KUKA KRL program: MyProgram_043().src

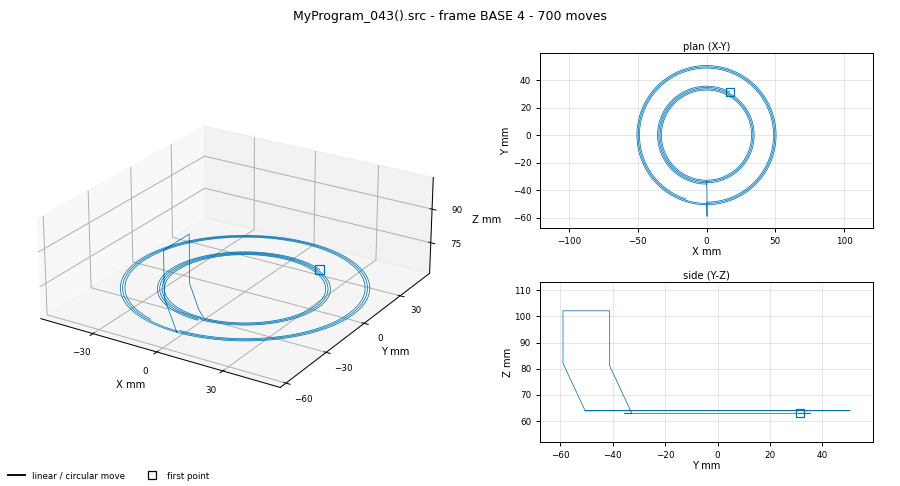
[picture p0: tool path of MyProgram_043().src in frame BASE 4, 700 of 700 moves have a stored position in this frame; points joined in program order, loops and branches not executed]
&ACCESS RVP
&REL 1
&PARAM TEMPLATE = C:\KRC\Roboter\Template\vorgabe
&PARAM EDITMASK = *
DEF MyProgram_043()
; ---- Setting reference (Base) ----
$BASE = BASE_DATA[4]

; --------------------------
; ---- Setting tool (TCP) ----
$TOOL = TOOL_DATA[3]
; --------------------------

$VEL.CP = VEL_APROX_PRINT
Startdeposition()
$VEL.CP = VEL_PRINT
LIN {X 16.8106,Y 31.3623,Z 63,A 55.0219,B 24.8198,C -3.0966,E1 25.0743,E2 -332.082} C_DIS
LIN {X 15.1626,Y 32.1914,Z 63,A 58.444,B 24.8186,C -3.1061,E1 25.0657,E2 -335.5177} C_DIS
LIN {X 13.6863,Y 32.8466,Z 63,A 60.9458,B 24.8184,C -3.1075,E1 25.0593,E2 -338.0168} C_DIS
LIN {X 11.5604,Y 33.654,Z 63,A 64.6472,B 24.818,C -3.1112,E1 25.0495,E2 -341.7194} C_DIS
LIN {X 8.9536,Y 34.4389,Z 63,A 68.8262,B 24.818,C -3.1115,E1 25.0383,E2 -345.8923} C_DIS
LIN {X 7.0657,Y 34.8749,Z 63,A 72.0407,B 24.8177,C -3.1142,E1 25.0295,E2 -349.1089} C_DIS
LIN {X 4.955,Y 35.237,Z 63,A 75.0597,B 24.8182,C -3.1099,E1 25.0213,E2 -352.1148} C_DIS
LIN {X 3.7288,Y 35.3877,Z 63,A 77.2434,B 24.8178,C -3.1126,E1 25.0152,E2 -354.3034} C_DIS
LIN {X 2.076,Y 35.5232,Z 63,A 79.8681,B 24.8179,C -3.1121,E1 25.0079,E2 -356.9257} C_DIS
LIN {X 0.3777,Y 35.582,Z 63,A 82.8072,B 24.8177,C -3.1142,E1 24.9997,E2 -359.8692} C_DIS
LIN {X -1.1222,Y 35.5659,Z 63,A 85.2424,B 24.8177,C -3.1138,E1 24.9929,E2 -362.3038} C_DIS
LIN {X -2.9049,Y 35.4649,Z 63,A 88.7717,B 24.817,C -3.1201,E1 24.983,E2 -365.8497} C_DIS
LIN {X -6.81,Y 34.926,Z 63,A 94.1207,B 24.8188,C -3.1045,E1 24.9683,E2 -371.1662} C_DIS
LIN {X -9.2966,Y 34.3477,Z 63,A 99.2069,B 24.818,C -3.1114,E1 24.9545,E2 -376.276} C_DIS
LIN {X -11.642,Y 33.6256,Z 63,A 102.3463,B 24.8196,C -3.098,E1 24.9462,E2 -379.3892} C_DIS
LIN {X -13.5299,Y 32.9112,Z 63,A 106.2069,B 24.8193,C -3.1002,E1 24.9362,E2 -383.2634} C_DIS
LIN {X -15.9173,Y 31.8253,Z 63,A 110.4655,B 24.82,C -3.0941,E1 24.9255,E2 -387.5184} C_DIS
LIN {X -18.0289,Y 30.6783,Z 63,A 114.2931,B 24.8208,C -3.087,E1 24.9162,E2 -391.3404} C_DIS
LIN {X -20.7669,Y 28.8954,Z 63,A 118.9134,B 24.8228,C -3.0705,E1 24.9056,E2 -395.9367} C_DIS
LIN {X -22.22,Y 27.7939,Z 63,A 122.3158,B 24.8229,C -3.069,E1 24.898,E2 -399.348} C_DIS
LIN {X -24.1802,Y 26.1054,Z 63,A 126.2379,B 24.8243,C -3.0574,E1 24.8899,E2 -403.2579} C_DIS
LIN {X -25.3409,Y 24.9807,Z 63,A 128.7227,B 24.8251,C -3.0502,E1 24.885,E2 -405.7359} C_DIS
LIN {X -26.8356,Y 23.3676,Z 63,A 133.3079,B 24.825,C -3.0515,E1 24.8764,E2 -410.3446} C_DIS
LIN {X -28.8287,Y 20.86,Z 63,A 137.8819,B 24.8271,C -3.0325,E1 24.8687,E2 -414.895} C_DIS
LIN {X -30.1785,Y 18.8534,Z 63,A 141.3427,B 24.8288,C -3.0179,E1 24.8635,E2 -418.3383} C_DIS
LIN {X -31.0448,Y 17.3901,Z 63,A 144.4056,B 24.8293,C -3.0132,E1 24.8592,E2 -421.4059} C_DIS
LIN {X -31.9505,Y 15.6632,Z 63,A 147.8398,B 24.8301,C -3.0068,E1 24.8549,E2 -424.8432} C_DIS
LIN {X -33.01,Y 13.2873,Z 63,A 152.0346,B 24.8315,C -2.9945,E1 24.8503,E2 -429.0318} C_DIS
LIN {X -33.7447,Y 11.2915,Z 63,A 155.0687,B 24.833,C -2.9806,E1 24.8475,E2 -432.0499} C_DIS
LIN {X -34.2032,Y 9.8157,Z 63,A 157.7943,B 24.8336,C -2.9752,E1 24.8454,E2 -434.7782} C_DIS
LIN {X -34.7895,Y 7.4763,Z 63,A 161.2013,B 24.8355,C -2.959,E1 24.8432,E2 -438.1663} C_DIS
LIN {X -35.0815,Y 5.9572,Z 63,A 164.5571,B 24.8355,C -2.9589,E1 24.8415,E2 -441.5418} C_DIS
LIN {X -35.4137,Y 3.4768,Z 63,A 168.3045,B 24.8372,C -2.9437,E1 24.8403,E2 -445.2754} C_DIS
LIN {X -35.5404,Y 1.7652,Z 63,A 171.2528,B 24.8379,C -2.9367,E1 24.8399,E2 -448.2247} C_DIS
LIN {X -35.5745,Y -0.8093,Z 63,A 174.7396,B 24.84,C -2.9179,E1 24.8399,E2 -451.6875} C_DIS
LIN {X -35.5121,Y -2.2598,Z 63,A 177.4397,B 24.8405,C -2.9139,E1 24.8402,E2 -454.3941} C_DIS
LIN {X -35.3438,Y -4.1241,Z 63,A -179.4444,B 24.8414,C -2.9055,E1 24.8411,E2 -457.5085} C_DIS
LIN {X -35.0507,Y -6.1346,Z 63,A -175.5471,B 24.8419,C -2.9011,E1 24.8429,E2 -461.4187} C_DIS
LIN {X -34.3748,Y -9.1965,Z 63,A -171.0715,B 24.8441,C -2.8808,E1 24.8458,E2 -465.8718} C_DIS
LIN {X -33.7609,Y -11.2432,Z 63,A -168.1618,B 24.8457,C -2.866,E1 24.8482,E2 -468.7628} C_DIS
LIN {X -33.2462,Y -12.6842,Z 63,A -165.0655,B 24.8458,C -2.8647,E1 24.8512,E2 -471.8735} C_DIS
LIN {X -32.3646,Y -14.7906,Z 63,A -161.0277,B 24.8466,C -2.8578,E1 24.8558,E2 -475.9171} C_DIS
LIN {X -31.2752,Y -16.9722,Z 63,A -157.1273,B 24.8477,C -2.8471,E1 24.8608,E2 -479.8126} C_DIS
LIN {X -30.1984,Y -18.8215,Z 63,A -153.4943,B 24.8485,C -2.8401,E1 24.8661,E2 -483.4474} C_DIS
LIN {X -28.8099,Y -20.8856,Z 63,A -150.0856,B 24.8501,C -2.8246,E1 24.8715,E2 -486.8358} C_DIS
LIN {X -27.7664,Y -22.253,Z 63,A -147.0838,B 24.8506,C -2.8204,E1 24.8767,E2 -489.8417} C_DIS
LIN {X -26.3842,Y -23.8768,Z 63,A -143.5764,B 24.8513,C -2.8135,E1 24.8832,E2 -493.3486} C_DIS
LIN {X -24.5192,Y -25.787,Z 63,A -139.4733,B 24.8524,C -2.8028,E1 24.8913,E2 -497.4433} C_DIS
LIN {X -23.1525,Y -27.0216,Z 63,A -136.4644,B 24.853,C -2.7976,E1 24.8976,E2 -500.4517} C_DIS
LIN {X -21.8431,Y -28.0903,Z 63,A -133.742,B 24.8535,C -2.7928,E1 24.9036,E2 -503.1727} C_DIS
LIN {X -20.5207,Y -29.0711,Z 63,A -130.4876,B 24.8533,C -2.7948,E1 24.911,E2 -506.4432} C_DIS
LIN {X -18.3593,Y -30.4819,Z 63,A -126.8445,B 24.8545,C -2.7832,E1 24.9196,E2 -510.0701} C_DIS
LIN {X -16.5344,Y -31.5089,Z 63,A -123.3892,B 24.8549,C -2.7797,E1 24.9281,E2 -513.5269} C_DIS
LIN {X -14.4801,Y -32.5045,Z 63,A -119.6559,B 24.8552,C -2.7763,E1 24.9375,E2 -517.2613} C_DIS
LIN {X -12.1069,Y -33.4608,Z 63,A -115.6723,B 24.8558,C -2.771,E1 24.9479,E2 -521.2407} C_DIS
LIN {X -10.7396,Y -33.9249,Z 63,A -113.2876,B 24.8558,C -2.7699,E1 24.9542,E2 -523.6272} C_DIS
LIN {X -8.9212,Y -34.4472,Z 63,A -110.3502,B 24.8562,C -2.7668,E1 24.9621,E2 -526.5618} C_DIS
LIN {X -7.1974,Y -34.8481,Z 63,A -107.4065,B 24.8562,C -2.7666,E1 24.9702,E2 -529.5087} C_DIS
LIN {X -5.1932,Y -35.2031,Z 63,A -104.0844,B 24.8562,C -2.7663,E1 24.9793,E2 -532.833} C_DIS
LIN {X -3.2172,Y -35.4379,Z 63,A -100.9818,B 24.8564,C -2.7647,E1 24.988,E2 -535.9337} C_DIS
LIN {X -1.3671,Y -35.5576,Z 63,A -98.1082,B 24.8565,C -2.7636,E1 24.996,E2 -538.8052} C_DIS
LIN {X 0.1757,Y -35.5825,Z 63,A -95.5141,B 24.8564,C -2.7655,E1 25.0032,E2 -541.4039} C_DIS
Enddeposition()
LIN {X 0.1757,Y -35.5825,Z 63,A -95.5141,B 24.8564,C -2.7655,E1 25.0032,E2 -541.4039} C_DIS
Startdeposition()
$VEL.CP = VEL_PRINT
LIN {X -0.0635,Y -34.634,Z 63,A -97.3781,B 24.8565,C -2.764,E1 24.998,E2 -539.5365} C_DIS
LIN {X -1.8941,Y -34.5819,Z 63,A -100.1272,B 24.8562,C -2.767,E1 24.9904,E2 -536.7939} C_DIS
LIN {X -3.4007,Y -34.467,Z 63,A -102.9968,B 24.8566,C -2.7628,E1 24.9823,E2 -533.9131} C_DIS
LIN {X -5.0318,Y -34.2667,Z 63,A -105.5259,B 24.8563,C -2.7655,E1 24.9754,E2 -531.3884} C_DIS
LIN {X -6.3765,Y -34.0415,Z 63,A -107.7692,B 24.8563,C -2.7664,E1 24.9692,E2 -529.1449} C_DIS
LIN {X -7.847,Y -33.7331,Z 63,A -110.4703,B 24.8563,C -2.7651,E1 24.9618,E2 -526.4375} C_DIS
LIN {X -10.2211,Y -33.0912,Z 63,A -113.9954,B 24.8555,C -2.7736,E1 24.9524,E2 -522.927} C_DIS
LIN {X -12.797,Y -32.1832,Z 63,A -119.1428,B 24.8558,C -2.7708,E1 24.9388,E2 -517.7624} C_DIS
LIN {X -14.7742,Y -31.325,Z 63,A -122.8072,B 24.8555,C -2.7736,E1 24.9295,E2 -514.0959} C_DIS
LIN {X -16.8249,Y -30.2725,Z 63,A -126.1313,B 24.8545,C -2.7834,E1 24.9213,E2 -510.7859} C_DIS
LIN {X -18.706,Y -29.1476,Z 63,A -130.3212,B 24.8545,C -2.783,E1 24.9113,E2 -506.5821} C_DIS
LIN {X -20.4124,Y -27.9792,Z 63,A -133.6933,B 24.8539,C -2.7891,E1 24.9037,E2 -503.2128} C_DIS
LIN {X -22.2197,Y -26.5668,Z 63,A -137.5576,B 24.8532,C -2.7952,E1 24.8953,E2 -499.3487} C_DIS
LIN {X -23.9602,Y -25.0084,Z 63,A -141.3526,B 24.8524,C -2.8035,E1 24.8875,E2 -495.5579} C_DIS
LIN {X -25.5766,Y -23.3526,Z 63,A -145.1707,B 24.8515,C -2.8117,E1 24.8802,E2 -491.7428} C_DIS
LIN {X -27.0497,Y -21.6299,Z 63,A -148.7189,B 24.8504,C -2.822,E1 24.8739,E2 -488.2029} C_DIS
LIN {X -28.2319,Y -20.0614,Z 63,A -152.2011,B 24.8498,C -2.8277,E1 24.8681,E2 -484.7175} C_DIS
LIN {X -29.5519,Y -18.0607,Z 63,A -155.8174,B 24.8484,C -2.8408,E1 24.8627,E2 -481.1142} C_DIS
LIN {X -30.3461,Y -16.6929,Z 63,A -159.348,B 24.8485,C -2.8396,E1 24.8578,E2 -477.5623} C_DIS
LIN {X -31.6295,Y -14.1099,Z 63,A -163.645,B 24.8467,C -2.8568,E1 24.8527,E2 -473.283} C_DIS
LIN {X -32.4602,Y -12.0779,Z 63,A -167.3733,B 24.8456,C -2.8662,E1 24.849,E2 -469.5563} C_DIS
LIN {X -33.016,Y -10.4631,Z 63,A -169.9052,B 24.8445,C -2.8769,E1 24.8468,E2 -467.0355} C_DIS
LIN {X -33.6352,Y -8.2566,Z 63,A -173.5321,B 24.8431,C -2.8896,E1 24.8441,E2 -463.4178} C_DIS
LIN {X -34.0004,Y -6.5934,Z 63,A -176.7425,B 24.8425,C -2.8948,E1 24.8423,E2 -460.201} C_DIS
LIN {X -34.2819,Y -4.9246,Z 63,A -179.5712,B 24.8416,C -2.9031,E1 24.8411,E2 -457.3753} C_DIS
LIN {X -34.5211,Y -2.7908,Z 63,A 176.9771,B 24.8403,C -2.9149,E1 24.8402,E2 -453.9312} C_DIS
LIN {X -34.6169,Y -1.0818,Z 63,A 174.3178,B 24.8392,C -2.9251,E1 24.8398,E2 -451.2804} C_DIS
LIN {X -34.6257,Y 0.7559,Z 63,A 170.7594,B 24.8386,C -2.9304,E1 24.8399,E2 -447.7131} C_DIS
LIN {X -34.5394,Y 2.5589,Z 63,A 168.2461,B 24.8372,C -2.9436,E1 24.8403,E2 -445.2163} C_DIS
LIN {X -34.342,Y 4.4866,Z 63,A 164.6999,B 24.8364,C -2.9508,E1 24.8415,E2 -441.6662} C_DIS
LIN {X -33.9758,Y 6.7211,Z 63,A 160.8095,B 24.8352,C -2.9613,E1 24.8434,E2 -437.7778} C_DIS
LIN {X -33.5133,Y 8.7391,Z 63,A 157.8409,B 24.8336,C -2.9756,E1 24.8453,E2 -434.8262} C_DIS
LIN {X -33.034,Y 10.4054,Z 63,A 154.5657,B 24.833,C -2.981,E1 24.848,E2 -431.5449} C_DIS
LIN {X -32.5136,Y 11.9319,Z 63,A 151.8111,B 24.8322,C -2.9883,E1 24.8505,E2 -428.7923} C_DIS
LIN {X -31.6838,Y 13.9879,Z 63,A 148.0384,B 24.831,C -2.9983,E1 24.8547,E2 -425.0225} C_DIS
LIN {X -30.8835,Y 15.6751,Z 63,A 144.9909,B 24.83,C -3.0075,E1 24.8584,E2 -421.9808} C_DIS
LIN {X -29.5734,Y 18.0254,Z 63,A 140.5667,B 24.8285,C -3.0203,E1 24.8646,E2 -417.564} C_DIS
LIN {X -28.3146,Y 19.9454,Z 63,A 136.653,B 24.8275,C -3.0295,E1 24.8707,E2 -413.653} C_DIS
LIN {X -26.9355,Y 21.771,Z 63,A 132.7973,B 24.8264,C -3.0387,E1 24.8774,E2 -409.801} C_DIS
LIN {X -25.4787,Y 23.4593,Z 63,A 129.2123,B 24.8253,C -3.0487,E1 24.884,E2 -406.2238} C_DIS
LIN {X -23.5824,Y 25.3655,Z 63,A 124.6722,B 24.8242,C -3.0581,E1 24.8931,E2 -401.6875} C_DIS
LIN {X -21.8898,Y 26.8393,Z 63,A 121.035,B 24.8232,C -3.0669,E1 24.9008,E2 -398.0572} C_DIS
LIN {X -20.1572,Y 28.1636,Z 63,A 117.5628,B 24.8222,C -3.0754,E1 24.9086,E2 -394.593} C_DIS
LIN {X -18.4097,Y 29.3358,Z 63,A 113.9792,B 24.8215,C -3.0809,E1 24.917,E2 -391.011} C_DIS
LIN {X -16.9995,Y 30.1747,Z 63,A 111.1515,B 24.8211,C -3.0846,E1 24.9238,E2 -388.1835} C_DIS
LIN {X -14.7244,Y 31.3481,Z 63,A 106.2891,B 24.8211,C -3.085,E1 24.9361,E2 -383.3096} C_DIS
LIN {X -11.4307,Y 32.6931,Z 63,A 101.432,B 24.819,C -3.103,E1 24.9486,E2 -378.4851} C_DIS
LIN {X -9.8087,Y 33.2158,Z 63,A 97.9102,B 24.8194,C -3.0989,E1 24.9581,E2 -374.9474} C_DIS
LIN {X -7.2365,Y 33.8696,Z 63,A 94.0249,B 24.8184,C -3.1082,E1 24.9686,E2 -371.0789} C_DIS
LIN {X -5.3631,Y 34.2161,Z 63,A 90.7464,B 24.8183,C -3.1091,E1 24.9776,E2 -367.7995} C_DIS
LIN {X -3.651,Y 34.4408,Z 63,A 87.6697,B 24.8183,C -3.1083,E1 24.9861,E2 -364.7188} C_DIS
LIN {X -2.1391,Y 34.568,Z 63,A 85.0882,B 24.8183,C -3.1085,E1 24.9933,E2 -362.1369} C_DIS
LIN {X 0.4092,Y 34.6319,Z 63,A 81.0243,B 24.818,C -3.1111,E1 25.0047,E2 -358.0793} C_DIS
LIN {X 1.9136,Y 34.5809,Z 63,A 78.6706,B 24.8178,C -3.1128,E1 25.0112,E2 -355.7303} C_DIS
LIN {X 3.832,Y 34.4215,Z 63,A 75.4828,B 24.8178,C -3.1124,E1 25.0201,E2 -352.5435} C_DIS
LIN {X 5.4581,Y 34.2012,Z 63,A 72.8563,B 24.8178,C -3.1127,E1 25.0273,E2 -349.9201} C_DIS
LIN {X 7.3944,Y 33.8352,Z 63,A 69.2492,B 24.8185,C -3.1072,E1 25.0372,E2 -346.3043} C_DIS
LIN {X 10.0204,Y 33.153,Z 63,A 64.8238,B 24.8187,C -3.105,E1 25.0491,E2 -341.8811} C_DIS
LIN {X 12.2173,Y 32.4074,Z 63,A 61.1221,B 24.8189,C -3.1034,E1 25.0588,E2 -338.183} C_DIS
LIN {X 14.2169,Y 31.5813,Z 63,A 57.0676,B 24.8201,C -3.0937,E1 25.0692,E2 -334.1152} C_DIS
LIN {X 16.87,Y 30.2473,Z 63,A 52.6482,B 24.8201,C -3.0936,E1 25.0801,E2 -329.7081} C_DIS
LIN {X 19.2374,Y 28.8,Z 63,A 48.2364,B 24.8206,C -3.089,E1 25.0905,E2 -325.2996} C_DIS
LIN {X 20.4873,Y 27.9243,Z 63,A 45.9769,B 24.8206,C -3.0883,E1 25.0957,E2 -323.0463} C_DIS
LIN {X 21.9684,Y 26.7745,Z 63,A 41.9109,B 24.8228,C -3.07,E1 25.1046,E2 -318.9521} C_DIS
LIN {X 23.9141,Y 25.0527,Z 63,A 37.7836,B 24.8235,C -3.0637,E1 25.113,E2 -314.8268} C_DIS
LIN {X 25.8678,Y 23.0296,Z 63,A 33.4254,B 24.8242,C -3.0577,E1 25.1213,E2 -310.4734} C_DIS
LIN {X 27.3526,Y 21.245,Z 63,A 29.6291,B 24.8252,C -3.0494,E1 25.1279,E2 -306.6751} C_DIS
LIN {X 28.3512,Y 19.893,Z 63,A 26.7406,B 24.8261,C -3.0412,E1 25.1326,E2 -303.7812} C_DIS
LIN {X 29.6598,Y 17.8833,Z 63,A 22.8855,B 24.8271,C -3.0326,E1 25.1383,E2 -299.9253} C_DIS
LIN {X 30.7733,Y 15.891,Z 63,A 19.1935,B 24.8281,C -3.0238,E1 25.1432,E2 -296.2318} C_DIS
LIN {X 31.7469,Y 13.8432,Z 63,A 16.033,B 24.8284,C -3.0219,E1 25.1469,E2 -293.0839} C_DIS
LIN {X 32.5142,Y 11.9303,Z 63,A 12.5189,B 24.8296,C -3.0107,E1 25.1505,E2 -289.5627} C_DIS
LIN {X 33.2079,Y 9.8352,Z 63,A 8.8585,B 24.8309,C -2.9999,E1 25.1536,E2 -285.8975} C_DIS
LIN {X 33.811,Y 7.5051,Z 63,A 4.497,B 24.8328,C -2.9825,E1 25.1565,E2 -281.5201} C_DIS
LIN {X 34.1619,Y 5.6977,Z 63,A 1.4153,B 24.8339,C -2.9727,E1 25.158,E2 -278.4332} C_DIS
LIN {X 34.5054,Y 2.9862,Z 63,A -3.0553,B 24.8354,C -2.9595,E1 25.1594,E2 -273.9578} C_DIS
LIN {X 34.6255,Y 0.7666,Z 63,A -6.5632,B 24.8364,C -2.9505,E1 25.1598,E2 -270.4494} C_DIS
LIN {X 34.5993,Y -1.5455,Z 63,A -10.4486,B 24.8378,C -2.9376,E1 25.1595,E2 -266.5566} C_DIS
LIN {X 34.4732,Y -3.3318,Z 63,A -12.9537,B 24.8381,C -2.935,E1 25.1589,E2 -264.0603} C_DIS
LIN {X 34.2793,Y -4.9431,Z 63,A -16.0017,B 24.8396,C -2.9213,E1 25.1578,E2 -260.9978} C_DIS
LIN {X 33.8998,Y -7.0921,Z 63,A -19.8009,B 24.8412,C -2.9073,E1 25.1558,E2 -257.1876} C_DIS
LIN {X 33.1911,Y -9.892,Z 63,A -24.2794,B 24.8423,C -2.897,E1 25.1525,E2 -252.7104} C_DIS
LIN {X 32.5177,Y -11.9206,Z 63,A -27.8522,B 24.8435,C -2.8857,E1 25.1492,E2 -249.1311} C_DIS
LIN {X 31.6889,Y -13.9762,Z 63,A -32.0187,B 24.8455,C -2.8676,E1 25.1446,E2 -244.9446} C_DIS
LIN {X 30.2023,Y -16.9506,Z 63,A -36.82,B 24.8461,C -2.8619,E1 25.1384,E2 -240.155} C_DIS
LIN {X 29.1784,Y -18.6581,Z 63,A -40.1878,B 24.8472,C -2.8516,E1 25.1335,E2 -236.7801} C_DIS
LIN {X 28.0786,Y -20.2752,Z 63,A -43.5148,B 24.8483,C -2.8416,E1 25.1281,E2 -233.4457} C_DIS
LIN {X 26.632,Y -22.1413,Z 63,A -47.8274,B 24.85,C -2.8259,E1 25.1205,E2 -229.1157} C_DIS
LIN {X 24.3949,Y -24.5844,Z 63,A -52.6985,B 24.8505,C -2.8211,E1 25.1112,E2 -224.2544} C_DIS
LIN {X 23.0523,Y -25.8475,Z 63,A -56.3973,B 24.8522,C -2.8052,E1 25.1035,E2 -220.5329} C_DIS
LIN {X 20.172,Y -28.153,Z 63,A -61.9593,B 24.8527,C -2.7999,E1 25.0912,E2 -214.9785} C_DIS
LIN {X 18.897,Y -29.0233,Z 63,A -64.7157,B 24.8535,C -2.7923,E1 25.0847,E2 -212.2132} C_DIS
LIN {X 16.4975,Y -30.4521,Z 63,A -68.7587,B 24.8535,C -2.7918,E1 25.075,E2 -208.1813} C_DIS
LIN {X 14.7635,Y -31.3299,Z 63,A -72.2932,B 24.8546,C -2.7825,E1 25.0661,E2 -204.6341} C_DIS
LIN {X 12.7079,Y -32.2182,Z 63,A -75.5559,B 24.8546,C -2.783,E1 25.0577,E2 -201.3803} C_DIS
LIN {X 10.6503,Y -32.9556,Z 63,A -79.8648,B 24.8559,C -2.7697,E1 25.0462,E2 -197.0483} C_DIS
LIN {X 8.7345,Y -33.5145,Z 63,A -82.4668,B 24.8553,C -2.7751,E1 25.0393,E2 -194.4632} C_DIS
LIN {X 7.1379,Y -33.8907,Z 63,A -85.5521,B 24.8561,C -2.768,E1 25.0308,E2 -191.3652} C_DIS
LIN {X 5.4364,Y -34.2044,Z 63,A -88.2199,B 24.8561,C -2.7682,E1 25.0235,E2 -188.7007} C_DIS
LIN {X 3.6386,Y -34.4421,Z 63,A -90.8735,B 24.8558,C -2.7706,E1 25.0162,E2 -186.0549} C_DIS
LIN {X 1.5293,Y -34.6,Z 63,A -95.3139,B 24.8571,C -2.7579,E1 25.0037,E2 -181.5861} C_DIS
LIN {X 1.5293,Y -34.6,Z 63,A -95.3139,B 24.8571,C -2.7579,E1 25.0037,E2 -181.5861} C_DIS
Enddeposition()
LIN {X 0.1418,Y -33.6777,Z 63,A -95.815,B 24.8533,C -2.7949,E1 25.0026,E2 -181.1731} C_DIS
Startdeposition()
$VEL.CP = VEL_PRINT
LIN {X 2.8514,Y -33.5634,Z 63,A -91.0405,B 24.8529,C -2.7986,E1 25.0159,E2 -185.9545} C_DIS
LIN {X 4.8668,Y -33.3307,Z 63,A -86.734,B 24.8515,C -2.8113,E1 25.0279,E2 -190.2875} C_DIS
LIN {X 7.9983,Y -32.7205,Z 63,A -81.8757,B 24.8518,C -2.809,E1 25.0411,E2 -195.134} C_DIS
LIN {X 10.4669,Y -32.0159,Z 63,A -77.9995,B 24.8519,C -2.8077,E1 25.0514,E2 -199.0004} C_DIS
LIN {X 11.957,Y -31.4903,Z 63,A -75.0907,B 24.8512,C -2.814,E1 25.0591,E2 -201.918} C_DIS
LIN {X 13.8798,Y -30.6914,Z 63,A -71.4979,B 24.8506,C -2.8198,E1 25.0683,E2 -205.5159} C_DIS
LIN {X 15.8468,Y -29.724,Z 63,A -67.6662,B 24.8498,C -2.8272,E1 25.0778,E2 -209.3547} C_DIS
LIN {X 17.6483,Y -28.6905,Z 63,A -64.1441,B 24.8492,C -2.8334,E1 25.0863,E2 -212.8807} C_DIS
LIN {X 19.2803,Y -27.6203,Z 63,A -60.9493,B 24.8487,C -2.8382,E1 25.0937,E2 -216.076} C_DIS
LIN {X 21.0567,Y -26.2918,Z 63,A -56.8255,B 24.8473,C -2.8509,E1 25.1028,E2 -220.2147} C_DIS
LIN {X 22.9024,Y -24.7006,Z 63,A -53.0751,B 24.8469,C -2.8548,E1 25.1106,E2 -223.9594} C_DIS
LIN {X 24.8683,Y -22.7196,Z 63,A -47.5228,B 24.8444,C -2.8776,E1 25.1213,E2 -229.5416} C_DIS
LIN {X 26.6927,Y -20.5452,Z 63,A -43.482,B 24.8443,C -2.8789,E1 25.1283,E2 -233.5666} C_DIS
LIN {X 28.2034,Y -18.416,Z 63,A -39.1453,B 24.8431,C -2.8895,E1 25.1352,E2 -237.907} C_DIS
LIN {X 29.378,Y -16.4786,Z 63,A -35.0709,B 24.8416,C -2.9035,E1 25.1409,E2 -241.9934} C_DIS
LIN {X 30.309,Y -14.6949,Z 63,A -31.8725,B 24.8409,C -2.9102,E1 25.1449,E2 -245.1907} C_DIS
LIN {X 31.2078,Y -12.6761,Z 63,A -28.104,B 24.8396,C -2.9214,E1 25.1491,E2 -248.9652} C_DIS
LIN {X 31.9406,Y -10.6963,Z 63,A -24.5863,B 24.8385,C -2.9312,E1 25.1523,E2 -252.4863} C_DIS
LIN {X 32.5772,Y -8.5655,Z 63,A -20.7114,B 24.8371,C -2.9442,E1 25.1552,E2 -256.3697} C_DIS
LIN {X 33.1042,Y -6.2243,Z 63,A -17.2808,B 24.8367,C -2.9474,E1 25.1572,E2 -259.7879} C_DIS
LIN {X 33.3154,Y -4.9723,Z 63,A -14.6256,B 24.8352,C -2.9613,E1 25.1584,E2 -262.4605} C_DIS
LIN {X 33.5534,Y -2.9655,Z 63,A -11.342,B 24.8342,C -2.9699,E1 25.1593,E2 -265.7449} C_DIS
LIN {X 33.6455,Y -1.6171,Z 63,A -8.8611,B 24.8331,C -2.9798,E1 25.1597,E2 -268.2345} C_DIS
LIN {X 33.6833,Y 0.1825,Z 63,A -5.9247,B 24.8323,C -2.9875,E1 25.1597,E2 -271.1718} C_DIS
LIN {X 33.6079,Y 2.2618,Z 63,A -2.4105,B 24.8311,C -2.9982,E1 25.1592,E2 -274.6902} C_DIS
LIN {X 33.4146,Y 4.2515,Z 63,A 0.9106,B 24.83,C -3.0075,E1 25.1582,E2 -278.0138} C_DIS
LIN {X 33.1059,Y 6.2155,Z 63,A 4.3752,B 24.8287,C -3.019,E1 25.1566,E2 -281.4854} C_DIS
LIN {X 32.4377,Y 9.0783,Z 63,A 9.8301,B 24.8262,C -3.0405,E1 25.1528,E2 -286.9597} C_DIS
LIN {X 31.5027,Y 11.9242,Z 63,A 14.2081,B 24.8257,C -3.0449,E1 25.1488,E2 -291.3234} C_DIS
LIN {X 30.9466,Y 13.302,Z 63,A 17.0215,B 24.8244,C -3.056,E1 25.1457,E2 -294.1478} C_DIS
LIN {X 30.0175,Y 15.2827,Z 63,A 20.6762,B 24.8234,C -3.0652,E1 25.1412,E2 -297.8046} C_DIS
LIN {X 28.9182,Y 17.2733,Z 63,A 24.9412,B 24.8216,C -3.0808,E1 25.1352,E2 -302.0848} C_DIS
LIN {X 27.6714,Y 19.2068,Z 63,A 28.1622,B 24.8216,C -3.0809,E1 25.1302,E2 -305.29} C_DIS
LIN {X 26.5354,Y 20.7488,Z 63,A 31.6472,B 24.8203,C -3.0917,E1 25.1243,E2 -308.784} C_DIS
LIN {X 25.1034,Y 22.4594,Z 63,A 35.6666,B 24.8189,C -3.1033,E1 25.1169,E2 -312.8127} C_DIS
LIN {X 23.582,Y 24.0522,Z 63,A 39.1309,B 24.8185,C -3.1072,E1 25.1101,E2 -316.2717} C_DIS
LIN {X 21.9707,Y 25.5328,Z 63,A 42.8867,B 24.8176,C -3.1148,E1 25.1023,E2 -320.0305} C_DIS
LIN {X 20.2752,Y 26.8985,Z 63,A 46.865,B 24.8164,C -3.125,E1 25.0935,E2 -324.0183} C_DIS
LIN {X 17.948,Y 28.504,Z 63,A 51.2457,B 24.8162,C -3.1269,E1 25.0833,E2 -328.3891} C_DIS
LIN {X 16.1698,Y 29.5493,Z 63,A 54.8034,B 24.8155,C -3.1323,E1 25.0746,E2 -331.9491} C_DIS
LIN {X 14.4618,Y 30.4217,Z 63,A 57.51,B 24.8159,C -3.1293,E1 25.0679,E2 -334.6412} C_DIS
LIN {X 13.009,Y 31.0705,Z 63,A 60.7616,B 24.8147,C -3.139,E1 25.0595,E2 -337.9079} C_DIS
LIN {X 10.9037,Y 31.8707,Z 63,A 64.6332,B 24.8143,C -3.1428,E1 25.0494,E2 -341.7807} C_DIS
LIN {X 8.7457,Y 32.5288,Z 63,A 68.6978,B 24.8136,C -3.1481,E1 25.0384,E2 -345.8512} C_DIS
LIN {X 6.1905,Y 33.1107,Z 63,A 72.9035,B 24.8138,C -3.1471,E1 25.027,E2 -350.0492} C_DIS
LIN {X 3.9481,Y 33.4518,Z 63,A 76.7395,B 24.8137,C -3.1477,E1 25.0163,E2 -353.8834} C_DIS
LIN {X 1.7512,Y 33.6386,Z 63,A 80.5794,B 24.8136,C -3.1488,E1 25.0057,E2 -357.7242} C_DIS
LIN {X -0.1115,Y 33.6838,Z 63,A 83.6232,B 24.8138,C -3.1469,E1 24.9972,E2 -360.7631} C_DIS
LIN {X -2.2988,Y 33.6054,Z 63,A 86.909,B 24.8145,C -3.1408,E1 24.988,E2 -364.0353} C_DIS
LIN {X -3.4658,Y 33.5052,Z 63,A 89.4035,B 24.814,C -3.1452,E1 24.9811,E2 -366.5417} C_DIS
LIN {X -5.8397,Y 33.1741,Z 63,A 93.1134,B 24.8148,C -3.1386,E1 24.9709,E2 -370.2391} C_DIS
LIN {X -7.6121,Y 32.8126,Z 63,A 96.5311,B 24.8147,C -3.1396,E1 24.9615,E2 -373.6632} C_DIS
LIN {X -9.762,Y 32.2389,Z 63,A 100.4078,B 24.815,C -3.1365,E1 24.9511,E2 -377.539} C_DIS
LIN {X -12.8437,Y 31.1395,Z 63,A 106.5675,B 24.8152,C -3.1353,E1 24.935,E2 -383.7088} C_DIS
LIN {X -15.1544,Y 30.0831,Z 63,A 110.2311,B 24.8167,C -3.1222,E1 24.9259,E2 -387.3505} C_DIS
LIN {X -17.0851,Y 29.0295,Z 63,A 114.0323,B 24.8174,C -3.1164,E1 24.9167,E2 -391.1489} C_DIS
LIN {X -18.9604,Y 27.841,Z 63,A 117.8358,B 24.8182,C -3.1095,E1 24.9078,E2 -394.9485} C_DIS
LIN {X -20.711,Y 26.5649,Z 63,A 121.5375,B 24.8191,C -3.1022,E1 24.8996,E2 -398.6459} C_DIS
LIN {X -22.3739,Y 25.18,Z 63,A 125.2495,B 24.82,C -3.0944,E1 24.8917,E2 -402.3539} C_DIS
LIN {X -24.0634,Y 23.5708,Z 63,A 129.6087,B 24.8207,C -3.0886,E1 24.8831,E2 -406.7176} C_DIS
LIN {X -25.8677,Y 21.5748,Z 63,A 133.749,B 24.8224,C -3.0734,E1 24.8755,E2 -410.8402} C_DIS
LIN {X -27.1512,Y 19.9354,Z 63,A 137.3212,B 24.8235,C -3.0644,E1 24.8695,E2 -414.408} C_DIS
LIN {X -28.3459,Y 18.1966,Z 63,A 140.9731,B 24.8245,C -3.0552,E1 24.8639,E2 -418.0563} C_DIS
LIN {X -29.5154,Y 16.2323,Z 63,A 145.3079,B 24.8254,C -3.0481,E1 24.8579,E2 -422.3966} C_DIS
LIN {X -30.5559,Y 14.1755,Z 63,A 148.6844,B 24.8272,C -3.0321,E1 24.8538,E2 -425.7532} C_DIS
LIN {X -31.3273,Y 12.3778,Z 63,A 152.0571,B 24.8283,C -3.0227,E1 24.8502,E2 -429.1218} C_DIS
LIN {X -32.1454,Y 10.0644,Z 63,A 156.4427,B 24.8295,C -3.0118,E1 24.8463,E2 -433.5065} C_DIS
LIN {X -32.7508,Y 7.8743,Z 63,A 160.2606,B 24.8309,C -2.9995,E1 24.8437,E2 -437.3172} C_DIS
LIN {X -33.1648,Y 5.8912,Z 63,A 163.7249,B 24.8321,C -2.989,E1 24.8418,E2 -440.7768} C_DIS
LIN {X -33.4765,Y 3.7371,Z 63,A 167.5749,B 24.8333,C -2.9786,E1 24.8405,E2 -444.6249} C_DIS
LIN {X -33.6543,Y 1.413,Z 63,A 171.4694,B 24.8347,C -2.9656,E1 24.8398,E2 -448.5118} C_DIS
LIN {X -33.6741,Y -0.8356,Z 63,A 174.965,B 24.8364,C -2.951,E1 24.8398,E2 -451.9934} C_DIS
LIN {X -33.5894,Y -2.5264,Z 63,A 178.3235,B 24.8369,C -2.946,E1 24.8405,E2 -455.3601} C_DIS
LIN {X -33.3483,Y -4.7435,Z 63,A -178.1101,B 24.8384,C -2.9324,E1 24.8417,E2 -458.9154} C_DIS
LIN {X -33.0657,Y -6.4236,Z 63,A -175.0144,B 24.8392,C -2.9253,E1 24.8433,E2 -462.0123} C_DIS
LIN {X -32.588,Y -8.5236,Z 63,A -171.229,B 24.8403,C -2.9154,E1 24.8458,E2 -465.7962} C_DIS
LIN {X -32.0009,Y -10.5154,Z 63,A -167.8181,B 24.8415,C -2.904,E1 24.8486,E2 -469.1994} C_DIS
LIN {X -31.2629,Y -12.5406,Z 63,A -164.0572,B 24.8426,C -2.8944,E1 24.8524,E2 -472.9586} C_DIS
LIN {X -30.42,Y -14.4655,Z 63,A -160.5273,B 24.8437,C -2.8842,E1 24.8565,E2 -476.4833} C_DIS
LIN {X -29.4147,Y -16.4129,Z 63,A -156.8425,B 24.8448,C -2.8739,E1 24.8613,E2 -480.163} C_DIS
LIN {X -28.3551,Y -18.1824,Z 63,A -152.9334,B 24.8454,C -2.8686,E1 24.8671,E2 -484.0793} C_DIS
LIN {X -26.9475,Y -20.2099,Z 63,A -148.9706,B 24.8467,C -2.8564,E1 24.8736,E2 -488.0321} C_DIS
LIN {X -25.5217,Y -21.9837,Z 63,A -145.0602,B 24.8476,C -2.8479,E1 24.8805,E2 -491.9404} C_DIS
LIN {X -24.0639,Y -23.5702,Z 63,A -141.3567,B 24.8484,C -2.8406,E1 24.8877,E2 -495.6424} C_DIS
LIN {X -22.4306,Y -25.1292,Z 63,A -137.54,B 24.8492,C -2.8328,E1 24.8955,E2 -499.4561} C_DIS
LIN {X -20.205,Y -26.9512,Z 63,A -133.1044,B 24.8506,C -2.8197,E1 24.9051,E2 -503.8769} C_DIS
LIN {X -19.0789,Y -27.7603,Z 63,A -130.3463,B 24.8506,C -2.8198,E1 24.9115,E2 -506.6447} C_DIS
LIN {X -17.5775,Y -28.7341,Z 63,A -127.169,B 24.851,C -2.8167,E1 24.919,E2 -509.8245} C_DIS
LIN {X -15.6236,Y -29.8415,Z 63,A -123.4867,B 24.8516,C -2.8103,E1 24.928,E2 -513.502} C_DIS
LIN {X -13.6792,Y -30.7818,Z 63,A -119.7679,B 24.852,C -2.8067,E1 24.9374,E2 -517.2215} C_DIS
LIN {X -11.7376,Y -31.5733,Z 63,A -115.8299,B 24.852,C -2.8073,E1 24.9477,E2 -521.1695} C_DIS
LIN {X -9.9843,Y -32.1702,Z 63,A -112.9773,B 24.8525,C -2.8018,E1 24.9553,E2 -524.014} C_DIS
LIN {X -7.8208,Y -32.7639,Z 63,A -108.9198,B 24.8525,C -2.8023,E1 24.9663,E2 -528.0787} C_DIS
LIN {X -5.5451,Y -33.2244,Z 63,A -105.2666,B 24.853,C -2.7977,E1 24.9763,E2 -531.7245} C_DIS
LIN {X -3.5533,Y -33.496,Z 63,A -101.601,B 24.8527,C -2.8,E1 24.9865,E2 -535.3981} C_DIS
LIN {X -0.965,Y -33.6702,Z 63,A -97.6474,B 24.8533,C -2.7949,E1 24.9975,E2 -539.3408} C_DIS
LIN {X 0.1418,Y -33.6777,Z 63,A -95.8149,B 24.8533,C -2.7949,E1 25.0026,E2 -541.1731} C_DIS
Enddeposition()
LIN {X 0.1418,Y -33.6777,Z 63,A -95.8149,B 24.8533,C -2.7949,E1 25.0026,E2 -541.1731} C_DIS
Startdeposition()
$VEL.CP = VEL_PRINT
LIN {X 0.0383,Y -32.7345,Z 63,A -97.4846,B 24.8533,C -2.7943,E1 24.9979,E2 -539.5021} C_DIS
LIN {X -2.0695,Y -32.6689,Z 63,A -101.2203,B 24.8534,C -2.7935,E1 24.9875,E2 -535.7635} C_DIS
LIN {X -4.6156,Y -32.407,Z 63,A -105.5946,B 24.8532,C -2.7953,E1 24.9754,E2 -531.3906} C_DIS
LIN {X -6.5528,Y -32.0715,Z 63,A -109.0641,B 24.8532,C -2.7962,E1 24.9658,E2 -527.9196} C_DIS
LIN {X -8.7368,Y -31.5472,Z 63,A -113.1573,B 24.8531,C -2.7968,E1 24.9548,E2 -523.8217} C_DIS
LIN {X -10.7999,Y -30.9012,Z 63,A -116.7946,B 24.8526,C -2.8012,E1 24.9451,E2 -520.1881} C_DIS
LIN {X -12.9003,Y -30.0856,Z 63,A -120.906,B 24.8524,C -2.8033,E1 24.9345,E2 -516.0727} C_DIS
LIN {X -15.0737,Y -29.0576,Z 63,A -125.1284,B 24.8519,C -2.8082,E1 24.9239,E2 -511.8509} C_DIS
LIN {X -17.1657,Y -27.8729,Z 63,A -129.2603,B 24.8512,C -2.8148,E1 24.914,E2 -507.7222} C_DIS
LIN {X -18.8505,Y -26.7622,Z 63,A -132.8134,B 24.8506,C -2.8202,E1 24.9058,E2 -504.17} C_DIS
LIN {X -20.5646,Y -25.468,Z 63,A -136.5377,B 24.8499,C -2.8271,E1 24.8976,E2 -500.4485} C_DIS
LIN {X -22.2854,Y -23.9774,Z 63,A -140.6726,B 24.8492,C -2.8334,E1 24.889,E2 -496.3122} C_DIS
LIN {X -23.9838,Y -22.2786,Z 63,A -144.9005,B 24.8483,C -2.842,E1 24.8808,E2 -492.0867} C_DIS
LIN {X -25.5531,Y -20.4597,Z 63,A -149.1286,B 24.8473,C -2.8513,E1 24.8733,E2 -487.8613} C_DIS
LIN {X -26.9845,Y -18.5308,Z 63,A -153.2535,B 24.8461,C -2.8621,E1 24.8666,E2 -483.7422} C_DIS
LIN {X -27.8655,Y -17.1776,Z 63,A -156.197,B 24.8454,C -2.8683,E1 24.8622,E2 -480.7985} C_DIS
LIN {X -28.9436,Y -15.2902,Z 63,A -159.8703,B 24.8442,C -2.8794,E1 24.8573,E2 -477.1324} C_DIS
LIN {X -29.9277,Y -13.2624,Z 63,A -164.0002,B 24.8432,C -2.8888,E1 24.8524,E2 -473.0023} C_DIS
LIN {X -30.8207,Y -11.0293,Z 63,A -168.2402,B 24.8419,C -2.9005,E1 24.8482,E2 -468.7666} C_DIS
LIN {X -31.5092,Y -8.8709,Z 63,A -171.9841,B 24.8405,C -2.9139,E1 24.8452,E2 -465.0331} C_DIS
LIN {X -32.001,Y -6.8894,Z 63,A -175.5891,B 24.8393,C -2.9243,E1 24.8429,E2 -461.4319} C_DIS
LIN {X -32.3829,Y -4.7853,Z 63,A -179.5953,B 24.8383,C -2.9337,E1 24.8411,E2 -457.4244} C_DIS
LIN {X -32.6462,Y -2.4056,Z 63,A 176.1793,B 24.8369,C -2.9464,E1 24.84,E2 -453.204} C_DIS
LIN {X -32.7333,Y -0.215,Z 63,A 172.4854,B 24.8354,C -2.9595,E1 24.8398,E2 -449.5192} C_DIS
LIN {X -32.6861,Y 1.772,Z 63,A 168.9651,B 24.8342,C -2.97,E1 24.8402,E2 -446.003} C_DIS
LIN {X -32.4877,Y 4.0136,Z 63,A 164.8389,B 24.833,C -2.9809,E1 24.8414,E2 -441.8782} C_DIS
LIN {X -32.1059,Y 6.3851,Z 63,A 160.6008,B 24.8315,C -2.9938,E1 24.8435,E2 -437.6457} C_DIS
LIN {X -31.5513,Y 8.7221,Z 63,A 156.366,B 24.8301,C -3.0065,E1 24.8464,E2 -433.4166} C_DIS
LIN {X -30.9097,Y 10.7757,Z 63,A 152.7126,B 24.8287,C -3.0187,E1 24.8496,E2 -429.7717} C_DIS
LIN {X -30.0871,Y 12.8967,Z 63,A 148.5611,B 24.8275,C -3.0292,E1 24.854,E2 -425.6221} C_DIS
LIN {X -29.1634,Y 14.8668,Z 63,A 144.886,B 24.8261,C -3.0413,E1 24.8585,E2 -421.9561} C_DIS
LIN {X -28.0729,Y 16.8365,Z 63,A 140.7614,B 24.825,C -3.0509,E1 24.8642,E2 -417.833} C_DIS
LIN {X -26.762,Y 18.8509,Z 63,A 136.5267,B 24.8237,C -3.062,E1 24.8708,E2 -413.6039} C_DIS
LIN {X -25.3066,Y 20.7638,Z 63,A 132.3223,B 24.8225,C -3.0729,E1 24.8781,E2 -409.4057} C_DIS
LIN {X -23.8361,Y 22.4357,Z 63,A 128.5752,B 24.8212,C -3.0836,E1 24.8851,E2 -405.6677} C_DIS
LIN {X -22.2736,Y 23.9885,Z 63,A 124.4967,B 24.8204,C -3.0907,E1 24.8933,E2 -401.5891} C_DIS
LIN {X -20.4536,Y 25.558,Z 63,A 120.267,B 24.8194,C -3.0995,E1 24.9024,E2 -397.3644} C_DIS
LIN {X -18.5233,Y 26.9897,Z 63,A 116.0396,B 24.8184,C -3.1076,E1 24.912,E2 -393.1417} C_DIS
LIN {X -16.6067,Y 28.2089,Z 63,A 112.292,B 24.8174,C -3.1168,E1 24.9209,E2 -389.4043} C_DIS
LIN {X -14.7148,Y 29.241,Z 63,A 108.3258,B 24.8168,C -3.1212,E1 24.9307,E2 -385.4376} C_DIS
LIN {X -12.7255,Y 30.1593,Z 63,A 104.5702,B 24.8161,C -3.1274,E1 24.9402,E2 -381.688} C_DIS
LIN {X -10.6308,Y 30.9603,Z 63,A 100.4779,B 24.8157,C -3.1308,E1 24.951,E2 -377.5954} C_DIS
LIN {X -8.3354,Y 31.6556,Z 63,A 96.2678,B 24.8152,C -3.135,E1 24.9623,E2 -373.3887} C_DIS
LIN {X -5.9936,Y 32.1813,Z 63,A 92.3698,B 24.8144,C -3.1414,E1 24.9729,E2 -369.5014} C_DIS
LIN {X -4.0311,Y 32.4854,Z 63,A 88.6371,B 24.8144,C -3.141,E1 24.9832,E2 -365.7649} C_DIS
LIN {X -1.9375,Y 32.677,Z 63,A 84.9198,B 24.8144,C -3.1422,E1 24.9936,E2 -362.0488} C_DIS
LIN {X 0.4201,Y 32.7319,Z 63,A 80.7761,B 24.8143,C -3.1429,E1 25.0051,E2 -357.9069} C_DIS
LIN {X 2.5829,Y 32.632,Z 63,A 77.1279,B 24.8141,C -3.1444,E1 25.0153,E2 -354.2637} C_DIS
LIN {X 4.8139,Y 32.3787,Z 63,A 73.0438,B 24.8144,C -3.1419,E1 25.0266,E2 -350.1769} C_DIS
LIN {X 7.1718,Y 31.9394,Z 63,A 69.0137,B 24.8144,C -3.1419,E1 25.0376,E2 -346.1519} C_DIS
LIN {X 9.1236,Y 31.4375,Z 63,A 65.3233,B 24.8149,C -3.1379,E1 25.0476,E2 -342.4577} C_DIS
LIN {X 11.4062,Y 30.6832,Z 63,A 61.1216,B 24.8153,C -3.1344,E1 25.0586,E2 -338.2562} C_DIS
LIN {X 13.6272,Y 29.7634,Z 63,A 56.9177,B 24.8158,C -3.1299,E1 25.0694,E2 -334.0519} C_DIS
LIN {X 15.7878,Y 28.6759,Z 63,A 52.8365,B 24.8162,C -3.1263,E1 25.0795,E2 -329.9736} C_DIS
LIN {X 17.5464,Y 27.6346,Z 63,A 49.3311,B 24.8167,C -3.122,E1 25.0878,E2 -326.4689} C_DIS
LIN {X 19.194,Y 26.5169,Z 63,A 45.7555,B 24.8175,C -3.1152,E1 25.096,E2 -322.8894} C_DIS
LIN {X 20.8703,Y 25.2181,Z 63,A 42.1027,B 24.8182,C -3.1092,E1 25.104,E2 -319.2362} C_DIS
LIN {X 22.5709,Y 23.709,Z 63,A 38.006,B 24.8193,C -3.0999,E1 25.1124,E2 -315.134} C_DIS
LIN {X 24.2456,Y 21.9934,Z 63,A 33.8619,B 24.8203,C -3.0916,E1 25.1203,E2 -310.9883} C_DIS
LIN {X 25.6828,Y 20.2957,Z 63,A 30.1585,B 24.8211,C -3.0852,E1 25.1269,E2 -307.2868} C_DIS
LIN {X 26.9916,Y 18.5206,Z 63,A 26.1983,B 24.8223,C -3.0745,E1 25.1333,E2 -303.3205} C_DIS
LIN {X 28.0838,Y 16.8183,Z 63,A 22.5982,B 24.8234,C -3.0646,E1 25.1386,E2 -299.7154} C_DIS
LIN {X 29.2414,Y 14.7139,Z 63,A 18.4187,B 24.8247,C -3.0537,E1 25.1441,E2 -295.5321} C_DIS
LIN {X 30.2419,Y 12.5295,Z 63,A 14.3754,B 24.8258,C -3.0442,E1 25.1486,E2 -291.4883} C_DIS
LIN {X 30.9623,Y 10.6249,Z 63,A 10.7122,B 24.8271,C -3.0327,E1 25.1521,E2 -287.8182} C_DIS
LIN {X 31.6523,Y 8.348,Z 63,A 6.5666,B 24.8285,C -3.0206,E1 25.1552,E2 -283.6678} C_DIS
LIN {X 32.1336,Y 6.2414,Z 63,A 2.9592,B 24.8295,C -3.0116,E1 25.1573,E2 -280.0602} C_DIS
LIN {X 32.4884,Y 4.0084,Z 63,A -1.1332,B 24.8311,C -2.9976,E1 25.1589,E2 -275.9587} C_DIS
LIN {X 32.6953,Y 1.6054,Z 63,A -5.3209,B 24.8325,C -2.985,E1 25.1597,E2 -271.7659} C_DIS
LIN {X 32.7247,Y -0.807,Z 63,A -9.4992,B 24.834,C -2.9724,E1 25.1597,E2 -267.5827} C_DIS
LIN {X 32.5818,Y -3.1576,Z 63,A -13.4944,B 24.8352,C -2.9612,E1 25.1588,E2 -263.5848} C_DIS
LIN {X 32.3171,Y -5.2116,Z 63,A -17.1134,B 24.8365,C -2.95,E1 25.1573,E2 -259.9605} C_DIS
LIN {X 31.9351,Y -7.1905,Z 63,A -20.7026,B 24.8378,C -2.9382,E1 25.1552,E2 -256.3642} C_DIS
LIN {X 31.3222,Y -9.512,Z 63,A -24.8796,B 24.8392,C -2.9256,E1 25.1521,E2 -252.1814} C_DIS
LIN {X 30.5401,Y -11.7839,Z 63,A -29.0572,B 24.8405,C -2.9133,E1 25.1481,E2 -247.9981} C_DIS
LIN {X 29.6356,Y -13.9019,Z 63,A -32.8816,B 24.8415,C -2.9043,E1 25.1437,E2 -244.1732} C_DIS
LIN {X 28.7212,Y -15.7043,Z 63,A -36.4884,B 24.8427,C -2.8932,E1 25.139,E2 -240.559} C_DIS
LIN {X 27.6411,Y -17.5362,Z 63,A -40.2674,B 24.8439,C -2.8821,E1 25.1335,E2 -236.7729} C_DIS
LIN {X 26.2881,Y -19.5062,Z 63,A -44.4282,B 24.8451,C -2.8712,E1 25.1267,E2 -232.6066} C_DIS
LIN {X 24.8271,Y -21.3344,Z 63,A -48.4129,B 24.8461,C -2.8622,E1 25.1196,E2 -228.6189} C_DIS
LIN {X 23.3896,Y -22.9013,Z 63,A -52.1291,B 24.847,C -2.8533,E1 25.1125,E2 -224.8977} C_DIS
LIN {X 21.7574,Y -24.457,Z 63,A -55.9604,B 24.8479,C -2.8457,E1 25.1046,E2 -221.0641} C_DIS
LIN {X 20.1308,Y -25.8129,Z 63,A -59.819,B 24.8489,C -2.8358,E1 25.0962,E2 -217.1966} C_DIS
LIN {X 18.1899,Y -27.2156,Z 63,A -63.9964,B 24.8498,C -2.8277,E1 25.0866,E2 -213.0144} C_DIS
LIN {X 16.3381,Y -28.3653,Z 63,A -67.6417,B 24.8503,C -2.823,E1 25.0779,E2 -209.3692} C_DIS
LIN {X 14.3498,Y -29.4218,Z 63,A -71.7242,B 24.8512,C -2.8149,E1 25.0677,E2 -205.2784} C_DIS
LIN {X 12.1523,Y -30.3954,Z 63,A -75.9054,B 24.8518,C -2.8092,E1 25.0569,E2 -201.0936} C_DIS
LIN {X 10.0211,Y -31.1625,Z 63,A -79.6995,B 24.8521,C -2.8064,E1 25.0469,E2 -197.3004} C_DIS
LIN {X 7.9122,Y -31.7639,Z 63,A -83.5811,B 24.8525,C -2.8019,E1 25.0364,E2 -193.4142} C_DIS
LIN {X 5.9733,Y -32.185,Z 63,A -87.1605,B 24.853,C -2.7978,E1 25.0266,E2 -189.8294} C_DIS
LIN {X 3.6101,Y -32.535,Z 63,A -91.3428,B 24.8532,C -2.7951,E1 25.015,E2 -185.6441} C_DIS
LIN {X 1.2286,Y -32.7115,Z 63,A -95.5167,B 24.8534,C -2.7935,E1 25.0034,E2 -181.468} C_DIS
LIN {X 1.2286,Y -32.7115,Z 63,A -95.5167,B 24.8534,C -2.7935,E1 25.0034,E2 -181.468} C_DIS
Enddeposition()
LIN {X 0.1644,Y -34.8455,Z 67.5315,A -95.5529,B 24.8518,C -2.8087,E1 25.0034,E2 -181.468} C_DIS
LIN {X 0.2867,Y -41.1836,Z 81.1262,A -95.5184,B 24.8533,C -2.7942,E1 25.0034,E2 -181.468} C_DIS
LIN {X 0.2867,Y -41.1836,Z 102.1262,A -95.8686,B 24.8374,C -2.9414,E1 25.0034,E2 -181.468} C_DIS
LIN {X 0.3916,Y -59.0086,Z 102.1262,A -95.4044,B 24.8688,C -2.6434,E1 25.0027,E2 -181.2233} C_DIS
LIN {X 0.3916,Y -59.0086,Z 82.1262,A -95.0713,B 24.8824,C -2.5033,E1 25.0027,E2 -181.2233} C_DIS
LIN {X 0.2964,Y -52.67,Z 68.5315,A -95.103,B 24.8811,C -2.5166,E1 25.0027,E2 -181.2233} C_DIS
LIN {X 0.2647,Y -50.5571,Z 64,A -95.115,B 24.8806,C -2.5217,E1 25.0027,E2 -181.2233} C_DIS
Startdeposition()
$VEL.CP = VEL_PRINT
LIN {X 2.8232,Y -50.4813,Z 64,A -92.015,B 24.8802,C -2.5263,E1 25.0114,E2 -184.3332} C_DIS
LIN {X 5.5729,Y -50.2521,Z 64,A -88.9538,B 24.8802,C -2.5267,E1 25.0199,E2 -187.3937} C_DIS
LIN {X 8.032,Y -49.919,Z 64,A -86.0255,B 24.8798,C -2.5308,E1 25.028,E2 -190.329} C_DIS
LIN {X 10.6138,Y -49.4339,Z 64,A -83.1233,B 24.8797,C -2.5319,E1 25.0359,E2 -193.2303} C_DIS
LIN {X 13.084,Y -48.838,Z 64,A -80.3136,B 24.8795,C -2.5335,E1 25.0435,E2 -196.0395} C_DIS
LIN {X 15.4418,Y -48.1446,Z 64,A -77.5409,B 24.8792,C -2.5365,E1 25.0509,E2 -198.8142} C_DIS
LIN {X 17.6787,Y -47.3693,Z 64,A -74.7599,B 24.8787,C -2.5418,E1 25.0583,E2 -201.602} C_DIS
LIN {X 20.0099,Y -46.4325,Z 64,A -71.9944,B 24.8785,C -2.5443,E1 25.0654,E2 -204.367} C_DIS
LIN {X 22.4595,Y -45.2979,Z 64,A -68.9662,B 24.8781,C -2.5485,E1 25.073,E2 -207.3972} C_DIS
LIN {X 24.6326,Y -44.1539,Z 64,A -66.1664,B 24.8776,C -2.5535,E1 25.0799,E2 -210.201} C_DIS
LIN {X 26.9409,Y -42.785,Z 64,A -63.1091,B 24.877,C -2.5594,E1 25.0872,E2 -213.2626} C_DIS
LIN {X 29.2417,Y -41.2465,Z 64,A -59.9761,B 24.8764,C -2.5655,E1 25.0944,E2 -216.3994} C_DIS
LIN {X 31.3588,Y -39.6605,Z 64,A -57.0229,B 24.8759,C -2.5709,E1 25.101,E2 -219.3547} C_DIS
LIN {X 33.3738,Y -37.9808,Z 64,A -54.0762,B 24.8753,C -2.577,E1 25.1072,E2 -222.3042} C_DIS
LIN {X 35.3104,Y -36.1879,Z 64,A -51.11,B 24.8747,C -2.5835,E1 25.1132,E2 -225.2735} C_DIS
LIN {X 37.1503,Y -34.2959,Z 64,A -48.14,B 24.874,C -2.5903,E1 25.1189,E2 -228.2469} C_DIS
LIN {X 38.8378,Y -32.3722,Z 64,A -45.227,B 24.8733,C -2.598,E1 25.1242,E2 -231.1647} C_DIS
LIN {X 40.5165,Y -30.2452,Z 64,A -42.1772,B 24.8725,C -2.6056,E1 25.1294,E2 -234.2182} C_DIS
LIN {X 42.0399,Y -28.0902,Z 64,A -39.1302,B 24.8716,C -2.6149,E1 25.1342,E2 -237.272} C_DIS
LIN {X 43.513,Y -25.7478,Z 64,A -36.0982,B 24.871,C -2.6216,E1 25.1386,E2 -240.3044} C_DIS
LIN {X 44.7433,Y -23.5449,Z 64,A -33.2735,B 24.8702,C -2.6291,E1 25.1424,E2 -243.1321} C_DIS
LIN {X 45.9171,Y -21.1657,Z 64,A -30.2237,B 24.8693,C -2.6388,E1 25.1461,E2 -246.1884} C_DIS
LIN {X 47.0104,Y -18.611,Z 64,A -27.1599,B 24.8685,C -2.6464,E1 25.1493,E2 -249.2534} C_DIS
LIN {X 47.8718,Y -16.2677,Z 64,A -24.359,B 24.8677,C -2.6545,E1 25.152,E2 -252.0575} C_DIS
LIN {X 48.6087,Y -13.9121,Z 64,A -21.5913,B 24.8669,C -2.6624,E1 25.1542,E2 -254.8284} C_DIS
LIN {X 49.2228,Y -11.5533,Z 64,A -18.8194,B 24.866,C -2.6712,E1 25.156,E2 -257.6051} C_DIS
LIN {X 49.7348,Y -9.0997,Z 64,A -16.0157,B 24.8652,C -2.6793,E1 25.1575,E2 -260.4115} C_DIS
LIN {X 50.1243,Y -6.6256,Z 64,A -13.1726,B 24.8643,C -2.6884,E1 25.1587,E2 -263.2593} C_DIS
LIN {X 50.4043,Y -3.9678,Z 64,A -10.1304,B 24.8633,C -2.6982,E1 25.1594,E2 -266.3067} C_DIS
LIN {X 50.545,Y -1.2408,Z 64,A -7.4894,B 24.8633,C -2.6985,E1 25.1598,E2 -268.9328} C_DIS
LIN {X 50.5568,Y 0.6205,Z 64,A -4.9307,B 24.8616,C -2.7145,E1 25.1598,E2 -271.514} C_DIS
LIN {X 50.4461,Y 3.3945,Z 64,A -1.8271,B 24.8607,C -2.7235,E1 25.1593,E2 -274.6203} C_DIS
LIN {X 50.1802,Y 6.1891,Z 64,A 1.2508,B 24.8599,C -2.7312,E1 25.1583,E2 -277.6982} C_DIS
LIN {X 49.8164,Y 8.644,Z 64,A 4.1582,B 24.8588,C -2.7418,E1 25.157,E2 -280.6136} C_DIS
LIN {X 49.3038,Y 11.2027,Z 64,A 7.0102,B 24.8581,C -2.7486,E1 25.1554,E2 -283.4652} C_DIS
LIN {X 48.6762,Y 13.6738,Z 64,A 9.8524,B 24.8573,C -2.7562,E1 25.1533,E2 -286.3091} C_DIS
LIN {X 47.9897,Y 15.9179,Z 64,A 12.5855,B 24.8563,C -2.7655,E1 25.151,E2 -289.0487} C_DIS
LIN {X 47.0632,Y 18.4766,Z 64,A 15.6449,B 24.8555,C -2.7739,E1 25.1479,E2 -292.1107} C_DIS
LIN {X 45.9678,Y 21.0548,Z 64,A 18.7273,B 24.8547,C -2.7809,E1 25.1445,E2 -295.1929} C_DIS
LIN {X 44.8794,Y 23.285,Z 64,A 21.4989,B 24.854,C -2.7877,E1 25.141,E2 -297.9658} C_DIS
LIN {X 43.6768,Y 25.4707,Z 64,A 24.4299,B 24.853,C -2.7972,E1 25.1369,E2 -300.9042} C_DIS
LIN {X 42.2128,Y 27.8283,Z 64,A 27.5289,B 24.8523,C -2.8043,E1 25.1323,E2 -304.0044} C_DIS
LIN {X 40.6506,Y 30.0653,Z 64,A 30.5519,B 24.8516,C -2.8104,E1 25.1273,E2 -307.0273} C_DIS
LIN {X 39.0465,Y 32.1211,Z 64,A 33.5376,B 24.8508,C -2.8179,E1 25.1221,E2 -310.0167} C_DIS
LIN {X 37.3337,Y 34.096,Z 64,A 36.4573,B 24.8502,C -2.8236,E1 25.1167,E2 -312.937} C_DIS
LIN {X 35.5193,Y 35.9821,Z 64,A 39.4324,B 24.8495,C -2.83,E1 25.1108,E2 -315.9145} C_DIS
LIN {X 33.5118,Y 37.8599,Z 64,A 42.5543,B 24.8489,C -2.8362,E1 25.1044,E2 -319.0386} C_DIS
LIN {X 31.47,Y 39.5726,Z 64,A 45.4842,B 24.8485,C -2.84,E1 25.0981,E2 -321.9664} C_DIS
LIN {X 29.3888,Y 41.1416,Z 64,A 48.4551,B 24.8479,C -2.8454,E1 25.0914,E2 -324.9394} C_DIS
LIN {X 27.1827,Y 42.6317,Z 64,A 51.4713,B 24.8474,C -2.8501,E1 25.0843,E2 -327.9568} C_DIS
LIN {X 24.913,Y 43.9973,Z 64,A 54.4512,B 24.847,C -2.8539,E1 25.0771,E2 -330.9367} C_DIS
LIN {X 22.6533,Y 45.2019,Z 64,A 57.4211,B 24.8464,C -2.8588,E1 25.0698,E2 -333.9102} C_DIS
LIN {X 20.3451,Y 46.2864,Z 64,A 60.2019,B 24.8464,C -2.86,E1 25.0627,E2 -336.6869} C_DIS
LIN {X 18.0268,Y 47.2375,Z 64,A 63.0674,B 24.846,C -2.8633,E1 25.0552,E2 -339.5536} C_DIS
LIN {X 15.6796,Y 48.0676,Z 64,A 65.8408,B 24.8458,C -2.8647,E1 25.0479,E2 -342.325} C_DIS
LIN {X 13.3223,Y 48.7736,Z 64,A 68.6219,B 24.8456,C -2.8665,E1 25.0405,E2 -345.1056} C_DIS
LIN {X 10.9241,Y 49.3662,Z 64,A 71.523,B 24.8453,C -2.8697,E1 25.0326,E2 -348.0105} C_DIS
LIN {X 8.377,Y 49.8614,Z 64,A 74.3946,B 24.8453,C -2.8696,E1 25.0247,E2 -350.8786} C_DIS
LIN {X 5.7294,Y 50.2347,Z 64,A 77.4903,B 24.8451,C -2.8714,E1 25.0161,E2 -353.976} C_DIS
LIN {X 3.0543,Y 50.4685,Z 64,A 80.5261,B 24.8451,C -2.8714,E1 25.0076,E2 -357.0104} C_DIS
LIN {X 0.3335,Y 50.5591,Z 64,A 83.5427,B 24.8453,C -2.8698,E1 24.9992,E2 -360.0227} C_DIS
LIN {X -2.254,Y 50.51,Z 64,A 86.4069,B 24.8455,C -2.8677,E1 24.9913,E2 -362.8825} C_DIS
LIN {X -4.7765,Y 50.3342,Z 64,A 89.4205,B 24.8454,C -2.8689,E1 24.9829,E2 -365.9003} C_DIS
LIN {X -7.444,Y 50.01,Z 64,A 92.3701,B 24.8457,C -2.8655,E1 24.9747,E2 -368.8439} C_DIS
LIN {X -10.0254,Y 49.5565,Z 64,A 95.3466,B 24.846,C -2.8633,E1 24.9665,E2 -371.8184} C_DIS
LIN {X -12.4379,Y 49.0067,Z 64,A 98.1871,B 24.8462,C -2.8613,E1 24.9588,E2 -374.6581} C_DIS
LIN {X -14.8529,Y 48.3295,Z 64,A 100.9216,B 24.8467,C -2.8565,E1 24.9515,E2 -377.3857} C_DIS
LIN {X -17.2047,Y 47.5431,Z 64,A 103.7496,B 24.847,C -2.8534,E1 24.9441,E2 -380.2117} C_DIS
LIN {X -19.4941,Y 46.6512,Z 64,A 106.6691,B 24.8472,C -2.8518,E1 24.9365,E2 -383.1338} C_DIS
LIN {X -21.8502,Y 45.595,Z 64,A 109.5782,B 24.8477,C -2.8471,E1 24.9292,E2 -386.0391} C_DIS
LIN {X -24.0705,Y 44.4628,Z 64,A 112.4185,B 24.8482,C -2.8428,E1 24.9221,E2 -388.8768} C_DIS
LIN {X -26.3006,Y 43.1812,Z 64,A 115.3459,B 24.8487,C -2.8378,E1 24.9151,E2 -391.8013} C_DIS
LIN {X -28.4757,Y 41.779,Z 64,A 118.3506,B 24.8492,C -2.8334,E1 24.9081,E2 -394.8053} C_DIS
LIN {X -30.6911,Y 40.18,Z 64,A 121.4213,B 24.8499,C -2.8267,E1 24.9013,E2 -397.8709} C_DIS
LIN {X -32.7708,Y 38.502,Z 64,A 124.4235,B 24.8506,C -2.8198,E1 24.8948,E2 -400.868} C_DIS
LIN {X -34.7181,Y 36.7559,Z 64,A 127.4299,B 24.8513,C -2.8137,E1 24.8886,E2 -403.8721} C_DIS
LIN {X -36.6184,Y 34.8636,Z 64,A 130.5354,B 24.8519,C -2.8074,E1 24.8826,E2 -406.9759} C_DIS
LIN {X -38.4163,Y 32.8714,Z 64,A 133.5555,B 24.8528,C -2.7996,E1 24.877,E2 -409.9909} C_DIS
LIN {X -40.0616,Y 30.8448,Z 64,A 136.5227,B 24.8536,C -2.792,E1 24.8719,E2 -412.954} C_DIS
LIN {X -41.5954,Y 28.7432,Z 64,A 139.4811,B 24.8544,C -2.7843,E1 24.8671,E2 -415.9084} C_DIS
LIN {X -43.045,Y 26.5236,Z 64,A 142.4658,B 24.8553,C -2.7757,E1 24.8627,E2 -418.8877} C_DIS
LIN {X -44.31,Y 24.3523,Z 64,A 145.3791,B 24.856,C -2.7686,E1 24.8587,E2 -421.7993} C_DIS
LIN {X -45.4837,Y 22.0819,Z 64,A 148.3008,B 24.8569,C -2.7606,E1 24.855,E2 -424.7176} C_DIS
LIN {X -46.5328,Y 19.775,Z 64,A 151.1884,B 24.8577,C -2.7523,E1 24.8518,E2 -427.6013} C_DIS
LIN {X -47.464,Y 17.4216,Z 64,A 154.0332,B 24.8586,C -2.7434,E1 24.849,E2 -430.4407} C_DIS
LIN {X -48.2557,Y 15.0909,Z 64,A 156.9535,B 24.8593,C -2.7368,E1 24.8464,E2 -433.3618} C_DIS
LIN {X -49.0211,Y 12.3816,Z 64,A 160.1311,B 24.8604,C -2.7267,E1 24.8442,E2 -436.534} C_DIS
LIN {X -49.6043,Y 9.7875,Z 64,A 163.1582,B 24.8613,C -2.7176,E1 24.8424,E2 -439.5569} C_DIS
LIN {X -50.0359,Y 7.2629,Z 64,A 166.0188,B 24.8623,C -2.7079,E1 24.8412,E2 -442.4114} C_DIS
LIN {X -50.3342,Y 4.7765,Z 64,A 168.9705,B 24.863,C -2.7006,E1 24.8403,E2 -445.3634} C_DIS
LIN {X -50.5201,Y 2.0184,Z 64,A 172.1408,B 24.864,C -2.6913,E1 24.8398,E2 -448.5304} C_DIS
LIN {X -50.5568,Y -0.6205,Z 64,A 175.1464,B 24.8649,C -2.6821,E1 24.8398,E2 -451.5322} C_DIS
LIN {X -50.4461,Y -3.3945,Z 64,A 178.2947,B 24.8659,C -2.6723,E1 24.8403,E2 -454.676} C_DIS
LIN {X -50.1802,Y -6.1891,Z 64,A -178.5682,B 24.867,C -2.6618,E1 24.8413,E2 -457.8068} C_DIS
LIN {X -49.8164,Y -8.644,Z 64,A -175.6352,B 24.8676,C -2.6549,E1 24.8426,E2 -460.7407} C_DIS
LIN {X -49.2971,Y -11.2315,Z 64,A -172.7302,B 24.8687,C -2.6446,E1 24.8443,E2 -463.6383} C_DIS
LIN {X -48.6762,Y -13.6738,Z 64,A -169.8624,B 24.8695,C -2.6363,E1 24.8463,E2 -466.5028} C_DIS
LIN {X -47.9256,Y -16.1082,Z 64,A -166.8587,B 24.8702,C -2.6296,E1 24.8489,E2 -469.5077} C_DIS
LIN {X -47.0038,Y -18.6275,Z 64,A -163.8052,B 24.871,C -2.6211,E1 24.8519,E2 -472.558} C_DIS
LIN {X -45.9171,Y -21.1657,Z 64,A -160.6418,B 24.8718,C -2.6129,E1 24.8555,E2 -475.7192} C_DIS
LIN {X -44.7355,Y -23.5598,Z 64,A -157.7052,B 24.8727,C -2.6034,E1 24.8593,E2 -478.6489} C_DIS
LIN {X -43.513,Y -25.7478,Z 64,A -154.7752,B 24.8733,C -2.5973,E1 24.8633,E2 -481.5796} C_DIS
LIN {X -42.0343,Y -28.0987,Z 64,A -151.5634,B 24.874,C -2.5903,E1 24.8682,E2 -484.7909} C_DIS
LIN {X -40.4557,Y -30.326,Z 64,A -148.5239,B 24.8748,C -2.5821,E1 24.8732,E2 -487.8255} C_DIS
LIN {X -38.8378,Y -32.3722,Z 64,A -145.5516,B 24.8755,C -2.5755,E1 24.8784,E2 -490.796} C_DIS
LIN {X -37.1126,Y -34.337,Z 64,A -142.5608,B 24.8761,C -2.5695,E1 24.884,E2 -493.7857} C_DIS
LIN {X -35.2862,Y -36.2118,Z 64,A -139.54,B 24.8766,C -2.5642,E1 24.89,E2 -496.8066} C_DIS
LIN {X -33.3653,Y -37.9882,Z 64,A -136.6083,B 24.8772,C -2.558,E1 24.8961,E2 -499.7352} C_DIS
LIN {X -31.3588,Y -39.6605,Z 64,A -133.5974,B 24.8776,C -2.5534,E1 24.9026,E2 -502.7465} C_DIS
LIN {X -29.1682,Y -41.299,Z 64,A -130.5394,B 24.8782,C -2.5476,E1 24.9095,E2 -505.8013} C_DIS
LIN {X -26.9165,Y -42.8002,Z 64,A -127.4088,B 24.8785,C -2.5439,E1 24.9169,E2 -508.9333} C_DIS
LIN {X -24.6326,Y -44.1539,Z 64,A -124.4804,B 24.879,C -2.5385,E1 24.9239,E2 -511.8575} C_DIS
LIN {X -22.4225,Y -45.3163,Z 64,A -121.5616,B 24.8792,C -2.5365,E1 24.9312,E2 -514.7794} C_DIS
LIN {X -19.9204,Y -46.4707,Z 64,A -118.4037,B 24.8795,C -2.5337,E1 24.9393,E2 -517.9383} C_DIS
LIN {X -17.4415,Y -47.4567,Z 64,A -115.468,B 24.8799,C -2.5295,E1 24.9469,E2 -520.8701} C_DIS
LIN {X -15.0909,Y -48.2557,Z 64,A -112.659,B 24.8801,C -2.5273,E1 24.9544,E2 -523.679} C_DIS
LIN {X -12.7325,Y -48.9309,Z 64,A -109.8862,B 24.8803,C -2.5255,E1 24.9618,E2 -526.4517} C_DIS
LIN {X -10.3175,Y -49.4965,Z 64,A -107.0542,B 24.8803,C -2.5246,E1 24.9696,E2 -529.2852} C_DIS
LIN {X -7.8764,Y -49.9431,Z 64,A -104.2244,B 24.8804,C -2.524,E1 24.9774,E2 -532.1164} C_DIS
LIN {X -5.3542,Y -50.276,Z 64,A -101.2714,B 24.8804,C -2.5249,E1 24.9856,E2 -535.0733} C_DIS
LIN {X -2.5931,Y -50.494,Z 64,A -98.1402,B 24.8804,C -2.5248,E1 24.9943,E2 -538.2055} C_DIS
LIN {X 0,Y -50.5611,Z 64,A -95.1269,B 24.8802,C -2.5267,E1 25.0027,E2 -541.2232} C_DIS
LIN {X 0,Y -50.5611,Z 64,A -95.1269,B 24.8802,C -2.5267,E1 25.0027,E2 -541.2232} C_DIS
Enddeposition()
LIN {X 0.2699,Y -49.6204,Z 64,A -96.2852,B 24.8811,C -2.5173,E1 24.9994,E2 -540.0428} C_DIS
Startdeposition()
$VEL.CP = VEL_PRINT
LIN {X -2.1675,Y -49.5741,Z 64,A -99.2436,B 24.8813,C -2.5145,E1 24.9911,E2 -537.0772} C_DIS
LIN {X -4.9328,Y -49.3756,Z 64,A -102.2913,B 24.8811,C -2.5172,E1 24.9827,E2 -534.0345} C_DIS
LIN {X -7.3165,Y -49.0798,Z 64,A -105.7396,B 24.8821,C -2.5066,E1 24.9731,E2 -530.5582} C_DIS
LIN {X -10.5954,Y -48.4771,Z 64,A -109.0953,B 24.8812,C -2.5162,E1 24.9639,E2 -527.2216} C_DIS
LIN {X -13.244,Y -47.8212,Z 64,A -112.1988,B 24.8809,C -2.5188,E1 24.9556,E2 -524.1197} C_DIS
LIN {X -15.761,Y -47.052,Z 64,A -116.1849,B 24.8821,C -2.506,E1 24.9449,E2 -520.0958} C_DIS
LIN {X -18.9909,Y -45.8439,Z 64,A -119.2486,B 24.8804,C -2.5243,E1 24.937,E2 -517.0689} C_DIS
LIN {X -21.4883,Y -44.7274,Z 64,A -122.4517,B 24.8801,C -2.5271,E1 24.9289,E2 -513.8645} C_DIS
LIN {X -24.0486,Y -43.4048,Z 64,A -125.5575,B 24.8794,C -2.5348,E1 24.9213,E2 -510.7684} C_DIS
LIN {X -26.041,Y -42.2398,Z 64,A -128.4468,B 24.8794,C -2.5351,E1 24.9143,E2 -507.871} C_DIS
LIN {X -28.2324,Y -40.8072,Z 64,A -131.4936,B 24.8789,C -2.5395,E1 24.9073,E2 -504.8245} C_DIS
LIN {X -30.6522,Y -39.0225,Z 64,A -134.4523,B 24.8776,C -2.5532,E1 24.9007,E2 -501.8879} C_DIS
LIN {X -31.8688,Y -38.0356,Z 64,A -136.9181,B 24.8783,C -2.5467,E1 24.8954,E2 -499.3972} C_DIS
LIN {X -34.0963,Y -36.052,Z 64,A -140.1883,B 24.8774,C -2.556,E1 24.8887,E2 -496.1359} C_DIS
LIN {X -35.9486,Y -34.2057,Z 64,A -143.2641,B 24.8768,C -2.5615,E1 24.8827,E2 -493.0601} C_DIS
LIN {X -37.7482,Y -32.2082,Z 64,A -146.4036,B 24.8762,C -2.5678,E1 24.8769,E2 -489.9217} C_DIS
LIN {X -39.4617,Y -30.0852,Z 64,A -149.599,B 24.8756,C -2.5745,E1 24.8714,E2 -486.7272} C_DIS
LIN {X -40.7366,Y -28.334,Z 64,A -151.9514,B 24.8748,C -2.5828,E1 24.8676,E2 -484.3829} C_DIS
LIN {X -42.0794,Y -26.2986,Z 64,A -155.0219,B 24.8744,C -2.5863,E1 24.8629,E2 -481.3052} C_DIS
LIN {X -43.4237,Y -24.0146,Z 64,A -157.9753,B 24.8735,C -2.5958,E1 24.8589,E2 -478.3591} C_DIS
LIN {X -44.668,Y -21.612,Z 64,A -161.1661,B 24.8728,C -2.6033,E1 24.8549,E2 -475.1693} C_DIS
LIN {X -45.7399,Y -19.2393,Z 64,A -164.1071,B 24.8718,C -2.6126,E1 24.8516,E2 -472.2343} C_DIS
LIN {X -46.9522,Y -16.056,Z 64,A -168.0406,B 24.8707,C -2.6239,E1 24.8478,E2 -468.3055} C_DIS
LIN {X -47.634,Y -13.9024,Z 64,A -170.7502,B 24.8701,C -2.6302,E1 24.8456,E2 -465.5953} C_DIS
LIN {X -48.3239,Y -11.2738,Z 64,A -173.9226,B 24.8692,C -2.6391,E1 24.8435,E2 -462.4258} C_DIS
LIN {X -49.044,Y -7.5484,Z 64,A -178.0524,B 24.8675,C -2.6559,E1 24.8415,E2 -458.3116} C_DIS
LIN {X -49.3269,Y -5.3968,Z 64,A 179.3028,B 24.867,C -2.6618,E1 24.8406,E2 -455.665} C_DIS
LIN {X -49.5239,Y -3.1114,Z 64,A 176.4245,B 24.8664,C -2.6669,E1 24.84,E2 -452.7817} C_DIS
LIN {X -49.6218,Y -0.198,Z 64,A 172.1105,B 24.8667,C -2.6648,E1 24.8398,E2 -448.4367} C_DIS
LIN {X -49.4199,Y 4.4688,Z 64,A 167.6479,B 24.8637,C -2.6942,E1 24.8407,E2 -444.0176} C_DIS
LIN {X -49.0902,Y 7.2452,Z 64,A 164.4523,B 24.8626,C -2.7048,E1 24.8418,E2 -440.8282} C_DIS
LIN {X -48.6255,Y 9.8925,Z 64,A 160.7123,B 24.8625,C -2.7059,E1 24.8438,E2 -437.0688} C_DIS
LIN {X -47.8179,Y 13.2562,Z 64,A 156.8911,B 24.861,C -2.7206,E1 24.8465,E2 -433.2603} C_DIS
LIN {X -46.8066,Y 16.4752,Z 64,A 153.3349,B 24.8593,C -2.737,E1 24.8496,E2 -429.7232} C_DIS
LIN {X -45.6792,Y 19.3827,Z 64,A 149.5702,B 24.8584,C -2.7455,E1 24.8536,E2 -425.9579} C_DIS
LIN {X -44.5253,Y 21.9037,Z 64,A 146.5374,B 24.8572,C -2.7572,E1 24.8572,E2 -422.9364} C_DIS
LIN {X -43.2926,Y 24.2497,Z 64,A 143.4551,B 24.8563,C -2.7656,E1 24.8613,E2 -419.858} C_DIS
LIN {X -41.9694,Y 26.4745,Z 64,A 140.2808,B 24.8557,C -2.7714,E1 24.8659,E2 -416.6811} C_DIS
LIN {X -40.6829,Y 28.4114,Z 64,A 137.9124,B 24.8545,C -2.783,E1 24.8696,E2 -414.3289} C_DIS
LIN {X -39.2823,Y 30.3182,Z 64,A 134.9479,B 24.8541,C -2.7869,E1 24.8746,E2 -411.3596} C_DIS
LIN {X -37.5204,Y 32.4737,Z 64,A 131.7125,B 24.8533,C -2.7948,E1 24.8804,E2 -408.128} C_DIS
LIN {X -35.6833,Y 34.4818,Z 64,A 128.3083,B 24.8529,C -2.7987,E1 24.887,E2 -404.7183} C_DIS
LIN {X -33.4438,Y 36.6582,Z 64,A 124.9231,B 24.8517,C -2.8101,E1 24.8938,E2 -401.3465} C_DIS
LIN {X -30.4879,Y 39.1515,Z 64,A 119.93,B 24.8515,C -2.812,E1 24.9047,E2 -396.3392} C_DIS
LIN {X -27.8901,Y 41.0419,Z 64,A 116.7669,B 24.8498,C -2.8273,E1 24.9118,E2 -393.2016} C_DIS
LIN {X -25.992,Y 42.2699,Z 64,A 114.3048,B 24.8491,C -2.8342,E1 24.9176,E2 -390.7484} C_DIS
LIN {X -23.9764,Y 43.445,Z 64,A 111.3945,B 24.8489,C -2.8356,E1 24.9247,E2 -387.833} C_DIS
LIN {X -21.5431,Y 44.7011,Z 64,A 108.2443,B 24.8484,C -2.8408,E1 24.9326,E2 -384.6867} C_DIS
LIN {X -19.1096,Y 45.7946,Z 64,A 105.1211,B 24.848,C -2.8446,E1 24.9406,E2 -381.5651} C_DIS
LIN {X -16.5999,Y 46.7625,Z 64,A 102.0753,B 24.8475,C -2.8494,E1 24.9485,E2 -378.5247} C_DIS
LIN {X -14.0401,Y 47.5932,Z 64,A 99.1407,B 24.8468,C -2.8556,E1 24.9563,E2 -375.5996} C_DIS
LIN {X -11.7581,Y 48.208,Z 64,A 96.1152,B 24.847,C -2.8536,E1 24.9645,E2 -372.565} C_DIS
LIN {X -9.0329,Y 48.793,Z 64,A 93.0716,B 24.8464,C -2.859,E1 24.9728,E2 -369.5307} C_DIS
LIN {X -6.8013,Y 49.1528,Z 64,A 90.0218,B 24.847,C -2.8537,E1 24.9813,E2 -366.4657} C_DIS
LIN {X -3.6916,Y 49.4847,Z 64,A 86.7589,B 24.8462,C -2.861,E1 24.9903,E2 -363.2185} C_DIS
LIN {X -1.2368,Y 49.606,Z 64,A 83.9351,B 24.8461,C -2.8621,E1 24.9982,E2 -360.3968} C_DIS
LIN {X 1.8092,Y 49.5889,Z 64,A 80.3087,B 24.8462,C -2.8608,E1 25.0083,E2 -356.7679} C_DIS
LIN {X 4.447,Y 49.4218,Z 64,A 76.6236,B 24.8474,C -2.8501,E1 25.0186,E2 -353.0593} C_DIS
LIN {X 7.5941,Y 49.0369,Z 64,A 73.6316,B 24.8463,C -2.8604,E1 25.0268,E2 -350.0944} C_DIS
LIN {X 10.3007,Y 48.5408,Z 64,A 70.313,B 24.8467,C -2.8566,E1 25.0359,E2 -346.771} C_DIS
LIN {X 13.8493,Y 47.6495,Z 64,A 65.9708,B 24.8472,C -2.852,E1 25.0477,E2 -342.4245} C_DIS
LIN {X 16.928,Y 46.6445,Z 64,A 62.3515,B 24.8472,C -2.8509,E1 25.0572,E2 -338.81} C_DIS
LIN {X 19.9321,Y 45.4422,Z 64,A 58.8732,B 24.8472,C -2.8517,E1 25.0661,E2 -335.3415} C_DIS
LIN {X 21.4629,Y 44.7397,Z 64,A 56.8428,B 24.8476,C -2.8479,E1 25.0713,E2 -333.3073} C_DIS
LIN {X 23.838,Y 43.521,Z 64,A 53.8009,B 24.848,C -2.8446,E1 25.0788,E2 -330.2662} C_DIS
LIN {X 26.1618,Y 42.1648,Z 64,A 50.6383,B 24.8486,C -2.8391,E1 25.0863,E2 -327.1004} C_DIS
LIN {X 28.5493,Y 40.5865,Z 64,A 47.7071,B 24.8484,C -2.8406,E1 25.0931,E2 -324.1828} C_DIS
LIN {X 29.6661,Y 39.777,Z 64,A 45.7782,B 24.8494,C -2.8317,E1 25.0975,E2 -322.2396} C_DIS
LIN {X 31.6738,Y 38.1977,Z 64,A 42.9675,B 24.8497,C -2.8289,E1 25.1036,E2 -319.4329} C_DIS
LIN {X 33.4959,Y 36.6102,Z 64,A 40.2385,B 24.8501,C -2.8247,E1 25.1092,E2 -316.7047} C_DIS
LIN {X 34.9536,Y 35.2214,Z 64,A 37.7641,B 24.8509,C -2.8171,E1 25.1142,E2 -314.2226} C_DIS
LIN {X 36.8368,Y 33.2472,Z 64,A 34.5933,B 24.8517,C -2.8099,E1 25.1202,E2 -311.0486} C_DIS
LIN {X 38.8025,Y 30.9303,Z 64,A 31.331,B 24.852,C -2.8065,E1 25.126,E2 -307.7935} C_DIS
LIN {X 40.3845,Y 28.8337,Z 64,A 28.1013,B 24.8532,C -2.7954,E1 25.1314,E2 -304.5531} C_DIS
LIN {X 41.8079,Y 26.7283,Z 64,A 25.2494,B 24.8538,C -2.7897,E1 25.1358,E2 -301.7017} C_DIS
LIN {X 43.0881,Y 24.6114,Z 64,A 22.5672,B 24.8542,C -2.7856,E1 25.1396,E2 -299.0237} C_DIS
LIN {X 44.1971,Y 22.5589,Z 64,A 19.6677,B 24.8554,C -2.7744,E1 25.1434,E2 -296.1129} C_DIS
LIN {X 45.3585,Y 20.1216,Z 64,A 16.3779,B 24.8567,C -2.7624,E1 25.1472,E2 -292.8125} C_DIS
LIN {X 46.1855,Y 18.1437,Z 64,A 14.1413,B 24.8569,C -2.76,E1 25.1495,E2 -290.5827} C_DIS
LIN {X 47.1074,Y 15.5958,Z 64,A 10.975,B 24.8579,C -2.7502,E1 25.1524,E2 -287.411} C_DIS
LIN {X 48.2359,Y 11.6439,Z 64,A 6.188,B 24.8595,C -2.7352,E1 25.1559,E2 -282.6161} C_DIS
LIN {X 48.7856,Y 9.072,Z 64,A 3.2772,B 24.8602,C -2.7285,E1 25.1575,E2 -279.7064} C_DIS
LIN {X 49.201,Y 6.4462,Z 64,A 0.2545,B 24.8611,C -2.72,E1 25.1587,E2 -276.6813} C_DIS
LIN {X 49.5177,Y 3.2075,Z 64,A -3.0745,B 24.8614,C -2.7169,E1 25.1595,E2 -273.3647} C_DIS
LIN {X 49.6092,Y 1.116,Z 64,A -5.5754,B 24.8623,C -2.7076,E1 25.1598,E2 -270.8568} C_DIS
LIN {X 49.6106,Y -1.0453,Z 64,A -8.5405,B 24.8641,C -2.6903,E1 25.1597,E2 -267.8685} C_DIS
LIN {X 49.4144,Y -4.5287,Z 64,A -12.3168,B 24.8649,C -2.6827,E1 25.1589,E2 -264.0966} C_DIS
LIN {X 49.1106,Y -7.1024,Z 64,A -15.3244,B 24.8658,C -2.673,E1 25.1578,E2 -261.0837} C_DIS
LIN {X 48.6447,Y -9.798,Z 64,A -17.9196,B 24.8657,C -2.6744,E1 25.1566,E2 -258.5071} C_DIS
LIN {X 48.2609,Y -11.5398,Z 64,A -20.4854,B 24.8674,C -2.6578,E1 25.1549,E2 -255.917} C_DIS
LIN {X 47.5683,Y -14.1261,Z 64,A -23.6194,B 24.8684,C -2.6474,E1 25.1526,E2 -252.7764} C_DIS
LIN {X 46.7355,Y -16.6752,Z 64,A -26.6526,B 24.8692,C -2.6393,E1 25.1498,E2 -249.741} C_DIS
LIN {X 45.4965,Y -19.8078,Z 64,A -30.4525,B 24.8702,C -2.6294,E1 25.1458,E2 -245.9387} C_DIS
LIN {X 44.3783,Y -22.2011,Z 64,A -33.5964,B 24.8713,C -2.6186,E1 25.142,E2 -242.7862} C_DIS
LIN {X 42.3599,Y -25.8444,Z 64,A -37.9251,B 24.8717,C -2.6145,E1 25.136,E2 -238.4701} C_DIS
LIN {X 41.3175,Y -27.4806,Z 64,A -40.5682,B 24.873,C -2.6003,E1 25.132,E2 -235.8067} C_DIS
LIN {X 39.7462,Y -29.7077,Z 64,A -43.7361,B 24.8739,C -2.5915,E1 25.1268,E2 -232.6332} C_DIS
LIN {X 37.8646,Y -32.0714,Z 64,A -47.0837,B 24.8745,C -2.5853,E1 25.1209,E2 -229.2864} C_DIS
LIN {X 35.7812,Y -34.3803,Z 64,A -50.7418,B 24.8755,C -2.5751,E1 25.1139,E2 -225.6204} C_DIS
LIN {X 33.8235,Y -36.3086,Z 64,A -53.9029,B 24.8762,C -2.5679,E1 25.1075,E2 -222.4553} C_DIS
LIN {X 31.7722,Y -38.1159,Z 64,A -57.0315,B 24.8768,C -2.5615,E1 25.1009,E2 -219.3236} C_DIS
LIN {X 29.3528,Y -40.0088,Z 64,A -60.5781,B 24.8775,C -2.5541,E1 25.093,E2 -215.7725} C_DIS
LIN {X 26.9628,Y -41.6573,Z 64,A -63.9364,B 24.8782,C -2.5475,E1 25.0852,E2 -212.4097} C_DIS
LIN {X 24.5957,Y -43.0971,Z 64,A -67.0845,B 24.8786,C -2.5427,E1 25.0776,E2 -209.26} C_DIS
LIN {X 22.3073,Y -44.3248,Z 64,A -70.4952,B 24.8798,C -2.5301,E1 25.0691,E2 -205.829} C_DIS
LIN {X 18.4391,Y -46.0681,Z 64,A -74.7904,B 24.8795,C -2.5341,E1 25.0581,E2 -201.5534} C_DIS
LIN {X 16.1243,Y -46.929,Z 64,A -77.6841,B 24.8799,C -2.5297,E1 25.0505,E2 -198.6551} C_DIS
LIN {X 13.1884,Y -47.8367,Z 64,A -81.2527,B 24.8803,C -2.5254,E1 25.041,E2 -195.0825} C_DIS
LIN {X 10.6782,Y -48.459,Z 64,A -84.3386,B 24.8807,C -2.5208,E1 25.0326,E2 -191.9901} C_DIS
LIN {X 7.977,Y -48.9765,Z 64,A -87.4235,B 24.8808,C -2.5199,E1 25.0241,E2 -188.9065} C_DIS
LIN {X 5.4536,Y -49.3208,Z 64,A -90.9427,B 24.8819,C -2.5081,E1 25.0143,E2 -185.3618} C_DIS
LIN {X 1.6411,Y -49.5945,Z 64,A -94.8446,B 24.8813,C -2.5151,E1 25.0034,E2 -181.478} C_DIS
LIN {X 1.6411,Y -49.5945,Z 64,A -94.8446,B 24.8813,C -2.5151,E1 25.0034,E2 -181.478} C_DIS
Enddeposition()
LIN {X 0.2772,Y -48.6819,Z 64,A -96.4414,B 24.8798,C -2.5309,E1 24.9991,E2 -179.9188} C_DIS
Startdeposition()
$VEL.CP = VEL_PRINT
LIN {X 1.8936,Y -48.6463,Z 64,A -92.4972,B 24.8763,C -2.5665,E1 25.0103,E2 -183.9468} C_DIS
LIN {X 5.1544,Y -48.4091,Z 64,A -89.4323,B 24.8775,C -2.5547,E1 25.0188,E2 -186.982} C_DIS
LIN {X 7.5029,Y -48.1012,Z 64,A -86.0483,B 24.8763,C -2.5672,E1 25.0282,E2 -190.3925} C_DIS
LIN {X 10.7195,Y -47.4882,Z 64,A -82.0725,B 24.8757,C -2.5727,E1 25.0391,E2 -194.3764} C_DIS
LIN {X 14.751,Y -46.394,Z 64,A -77.6975,B 24.8762,C -2.5683,E1 25.0507,E2 -198.7333} C_DIS
LIN {X 17.2598,Y -45.5205,Z 64,A -74.6936,B 24.876,C -2.5701,E1 25.0586,E2 -201.7353} C_DIS
LIN {X 19.9642,Y -44.4008,Z 64,A -70.9333,B 24.8749,C -2.5809,E1 25.0683,E2 -205.5122} C_DIS
LIN {X 22.1315,Y -43.3613,Z 64,A -68.0837,B 24.8745,C -2.5858,E1 25.0754,E2 -208.3658} C_DIS
LIN {X 25.1788,Y -41.666,Z 64,A -64.4665,B 24.8747,C -2.5839,E1 25.0841,E2 -211.9677} C_DIS
LIN {X 27.1702,Y -40.3957,Z 64,A -61.4408,B 24.8737,C -2.5939,E1 25.0912,E2 -215.007} C_DIS
LIN {X 29.5405,Y -38.6965,Z 64,A -58.3324,B 24.8736,C -2.5947,E1 25.0982,E2 -218.1064} C_DIS
LIN {X 32.1929,Y -36.5194,Z 64,A -54.0251,B 24.8722,C -2.6087,E1 25.1075,E2 -222.4302} C_DIS
LIN {X 34.1709,Y -34.6751,Z 64,A -50.4503,B 24.8707,C -2.6238,E1 25.1147,E2 -226.0258} C_DIS
LIN {X 36.8153,Y -31.854,Z 64,A -46.6364,B 24.871,C -2.6207,E1 25.1218,E2 -229.8154} C_DIS
LIN {X 38.1777,Y -30.2072,Z 64,A -43.8218,B 24.8698,C -2.633,E1 25.1268,E2 -232.6462} C_DIS
LIN {X 40.0457,Y -27.6833,Z 64,A -40.7541,B 24.8701,C -2.6306,E1 25.1318,E2 -235.6934} C_DIS
LIN {X 41.5167,Y -25.4241,Z 64,A -36.4839,B 24.867,C -2.6611,E1 25.1382,E2 -240.0142} C_DIS
LIN {X 43.2666,Y -22.3169,Z 64,A -32.7781,B 24.8668,C -2.6633,E1 25.1431,E2 -243.7058} C_DIS
LIN {X 44.2418,Y -20.3148,Z 64,A -30.084,B 24.8659,C -2.6725,E1 25.1463,E2 -246.4071} C_DIS
LIN {X 45.3567,Y -17.686,Z 64,A -26.8255,B 24.8651,C -2.6805,E1 25.1497,E2 -249.6665} C_DIS
LIN {X 46.2996,Y -15.0452,Z 64,A -23.592,B 24.8642,C -2.6892,E1 25.1527,E2 -252.9024} C_DIS
LIN {X 47.0571,Y -12.4751,Z 64,A -20.4609,B 24.8632,C -2.6985,E1 25.155,E2 -256.0375} C_DIS
LIN {X 47.7454,Y -9.5071,Z 64,A -16.9669,B 24.8623,C -2.7078,E1 25.1571,E2 -259.5333} C_DIS
LIN {X 48.2256,Y -6.6587,Z 64,A -13.6072,B 24.8613,C -2.7177,E1 25.1585,E2 -262.8966} C_DIS
LIN {X 48.5101,Y -4.0977,Z 64,A -10.5556,B 24.8603,C -2.7276,E1 25.1594,E2 -265.9536} C_DIS
LIN {X 48.6678,Y -1.2081,Z 64,A -7.1442,B 24.8592,C -2.7385,E1 25.1598,E2 -269.3703} C_DIS
LIN {X 48.6257,Y 2.3556,Z 64,A -3.3658,B 24.8587,C -2.7433,E1 25.1595,E2 -273.1376} C_DIS
LIN {X 48.2325,Y 6.6099,Z 64,A 2.0364,B 24.8563,C -2.7663,E1 25.158,E2 -278.5623} C_DIS
LIN {X 47.7895,Y 9.2836,Z 64,A 5.3815,B 24.8549,C -2.7792,E1 25.1563,E2 -281.9183} C_DIS
LIN {X 47.0826,Y 12.3783,Z 64,A 8.6822,B 24.8547,C -2.7817,E1 25.1541,E2 -285.2059} C_DIS
LIN {X 46.4423,Y 14.5987,Z 64,A 11.6089,B 24.8534,C -2.7938,E1 25.1518,E2 -288.1446} C_DIS
LIN {X 45.5323,Y 17.2286,Z 64,A 14.423,B 24.8534,C -2.7942,E1 25.1491,E2 -290.9437} C_DIS
LIN {X 44.4305,Y 19.8982,Z 64,A 18.361,B 24.8512,C -2.8143,E1 25.1448,E2 -294.9078} C_DIS
LIN {X 43.1878,Y 22.4685,Z 64,A 21.559,B 24.8506,C -2.8203,E1 25.1408,E2 -298.1029} C_DIS
LIN {X 41.1603,Y 25.9971,Z 64,A 26.2477,B 24.8495,C -2.8307,E1 25.1341,E2 -302.7922} C_DIS
LIN {X 39.6354,Y 28.2673,Z 64,A 29.9277,B 24.8477,C -2.8476,E1 25.1282,E2 -306.4941} C_DIS
LIN {X 37.3181,Y 31.2633,Z 64,A 33.9888,B 24.8474,C -2.8503,E1 25.1212,E2 -310.5427} C_DIS
LIN {X 35.5222,Y 33.2895,Z 64,A 37.1869,B 24.8466,C -2.8575,E1 25.1151,E2 -313.7437} C_DIS
LIN {X 33.63,Y 35.2004,Z 64,A 40.8108,B 24.845,C -2.8727,E1 25.1078,E2 -317.3884} C_DIS
LIN {X 31.0086,Y 37.53,Z 64,A 44.4208,B 24.8452,C -2.8707,E1 25.1002,E2 -320.9797} C_DIS
LIN {X 28.8306,Y 39.2278,Z 64,A 47.3416,B 24.8452,C -2.8703,E1 25.0938,E2 -323.8889} C_DIS
LIN {X 27.4734,Y 40.1901,Z 64,A 50.1679,B 24.8431,C -2.8895,E1 25.0872,E2 -326.7511} C_DIS
LIN {X 24.3537,Y 42.1535,Z 64,A 53.9667,B 24.8435,C -2.8859,E1 25.0781,E2 -330.5295} C_DIS
LIN {X 21.9229,Y 43.4672,Z 64,A 57.0854,B 24.8433,C -2.8876,E1 25.0704,E2 -333.6437} C_DIS
LIN {X 18.6754,Y 44.9585,Z 64,A 61.0174,B 24.8433,C -2.8874,E1 25.0604,E2 -337.5654} C_DIS
LIN {X 15.8134,Y 46.0432,Z 64,A 64.7896,B 24.8427,C -2.8936,E1 25.0505,E2 -341.3445} C_DIS
LIN {X 13.4052,Y 46.8009,Z 64,A 68.0422,B 24.8419,C -2.9006,E1 25.0418,E2 -344.608} C_DIS
LIN {X 10.9612,Y 47.4327,Z 64,A 70.9308,B 24.8419,C -2.9008,E1 25.034,E2 -347.4929} C_DIS
LIN {X 8.1666,Y 47.9928,Z 64,A 74.0116,B 24.8423,C -2.8975,E1 25.0255,E2 -350.5622} C_DIS
LIN {X 6.7325,Y 48.2151,Z 64,A 76.27,B 24.8412,C -2.9072,E1 25.0192,E2 -352.8418} C_DIS
LIN {X 2.5483,Y 48.6162,Z 64,A 80.6907,B 24.8421,C -2.8986,E1 25.007,E2 -357.2399} C_DIS
LIN {X -0.7144,Y 48.6775,Z 64,A 84.7728,B 24.8418,C -2.902,E1 24.9956,E2 -361.3295} C_DIS
LIN {X -3.4098,Y 48.5633,Z 64,A 87.9119,B 24.842,C -2.9002,E1 24.9868,E2 -364.4653} C_DIS
LIN {X -6.6805,Y 48.2225,Z 64,A 92.2724,B 24.8413,C -2.9059,E1 24.9747,E2 -368.8424} C_DIS
LIN {X -10.5903,Y 47.517,Z 64,A 96.5123,B 24.8425,C -2.8952,E1 24.9632,E2 -373.0616} C_DIS
LIN {X -12.9336,Y 46.9332,Z 64,A 99.3261,B 24.8429,C -2.8919,E1 24.9556,E2 -375.8719} C_DIS
LIN {X -15.525,Y 46.141,Z 64,A 102.5637,B 24.8432,C -2.889,E1 24.947,E2 -379.1083} C_DIS
LIN {X -18.0765,Y 45.2021,Z 64,A 105.6259,B 24.8439,C -2.8827,E1 24.939,E2 -382.1621} C_DIS
LIN {X -20.4515,Y 44.1787,Z 64,A 108.8265,B 24.8441,C -2.8807,E1 24.9308,E2 -385.3655} C_DIS
LIN {X -22.854,Y 42.9854,Z 64,A 111.9631,B 24.8447,C -2.8753,E1 24.9231,E2 -388.4978} C_DIS
LIN {X -24.5521,Y 42.0389,Z 64,A 114.6788,B 24.8444,C -2.8777,E1 24.9165,E2 -391.2273} C_DIS
LIN {X -27.6745,Y 40.0518,Z 64,A 118.4318,B 24.8463,C -2.8605,E1 24.9078,E2 -394.9516} C_DIS
LIN {X -30.0017,Y 38.34,Z 64,A 122.4883,B 24.846,C -2.8632,E1 24.8987,E2 -399.0291} C_DIS
LIN {X -32.5933,Y 36.1623,Z 64,A 125.9801,B 24.8477,C -2.8472,E1 24.8914,E2 -402.4965} C_DIS
LIN {X -35.5587,Y 33.2507,Z 64,A 130.9673,B 24.8488,C -2.837,E1 24.8816,E2 -407.4805} C_DIS
LIN {X -37.3499,Y 31.2253,Z 64,A 134.2158,B 24.8495,C -2.83,E1 24.8757,E2 -410.7269} C_DIS
LIN {X -39.0024,Y 29.1349,Z 64,A 137.2286,B 24.8506,C -2.8201,E1 24.8706,E2 -413.7304} C_DIS
LIN {X -40.5543,Y 26.9329,Z 64,A 141.2023,B 24.8503,C -2.8227,E1 24.8644,E2 -417.7302} C_DIS
LIN {X -42.5633,Y 23.6304,Z 64,A 145.0849,B 24.8527,C -2.8006,E1 24.859,E2 -421.5802} C_DIS
LIN {X -43.7343,Y 21.385,Z 64,A 147.7801,B 24.854,C -2.7881,E1 24.8556,E2 -424.2598} C_DIS
LIN {X -44.5403,Y 19.6505,Z 64,A 150.4559,B 24.854,C -2.7873,E1 24.8525,E2 -426.9484} C_DIS
LIN {X -45.6092,Y 17.0254,Z 64,A 153.3471,B 24.8557,C -2.7712,E1 24.8495,E2 -429.8173} C_DIS
LIN {X -46.3839,Y 14.7831,Z 64,A 156.8312,B 24.8557,C -2.7722,E1 24.8465,E2 -433.3236} C_DIS
LIN {X -47.3454,Y 11.3311,Z 64,A 160.8266,B 24.8573,C -2.7561,E1 24.8437,E2 -437.3039} C_DIS
LIN {X -47.9144,Y 8.615,Z 64,A 163.9069,B 24.8586,C -2.7434,E1 24.842,E2 -440.372} C_DIS
LIN {X -48.3046,Y 6.0593,Z 64,A 167.2082,B 24.8593,C -2.7374,E1 24.8407,E2 -443.6786} C_DIS
LIN {X -48.5243,Y 3.9252,Z 64,A 169.9956,B 24.8597,C -2.733,E1 24.8401,E2 -446.4723} C_DIS
LIN {X -48.6791,Y 0.5401,Z 64,A 173.3767,B 24.8618,C -2.7123,E1 24.8398,E2 -449.8241} C_DIS
LIN {X -48.6495,Y -1.8013,Z 64,A 176.9206,B 24.8616,C -2.7143,E1 24.8401,E2 -453.3942} C_DIS
LIN {X -48.3334,Y -5.821,Z 64,A -178.775,B 24.8637,C -2.6936,E1 24.8412,E2 -457.6748} C_DIS
LIN {X -48.0597,Y -7.767,Z 64,A -175.9581,B 24.8637,C -2.6934,E1 24.8424,E2 -460.5081} C_DIS
LIN {X -47.4023,Y -11.093,Z 64,A -172.397,B 24.8656,C -2.6754,E1 24.8445,E2 -464.0471} C_DIS
LIN {X -46.7647,Y -13.53,Z 64,A -169.7776,B 24.8669,C -2.6619,E1 24.8464,E2 -466.6493} C_DIS
LIN {X -46.0683,Y -15.7396,Z 64,A -166.1748,B 24.8665,C -2.6661,E1 24.8496,E2 -470.2827} C_DIS
LIN {X -44.4354,Y -19.8871,Z 64,A -161.3804,B 24.8686,C -2.6449,E1 24.8547,E2 -475.0533} C_DIS
LIN {X -43.2766,Y -22.2974,Z 64,A -157.8181,B 24.8689,C -2.6423,E1 24.8592,E2 -478.6284} C_DIS
LIN {X -41.5248,Y -25.4109,Z 64,A -153.943,B 24.8705,C -2.6266,E1 24.8647,E2 -482.4862} C_DIS
LIN {X -40.0632,Y -27.6582,Z 64,A -150.8591,B 24.8713,C -2.6178,E1 24.8695,E2 -485.5643} C_DIS
LIN {X -38.0022,Y -30.4288,Z 64,A -146.7116,B 24.8722,C -2.6094,E1 24.8765,E2 -489.7115} C_DIS
LIN {X -36.2983,Y -32.4415,Z 64,A -143.592,B 24.8728,C -2.6027,E1 24.8822,E2 -492.8293} C_DIS
LIN {X -34.4332,Y -34.4158,Z 64,A -140.3584,B 24.8734,C -2.5966,E1 24.8885,E2 -496.0621} C_DIS
LIN {X -31.8054,Y -36.8574,Z 64,A -136.0765,B 24.8741,C -2.5893,E1 24.8974,E2 -500.3437} C_DIS
LIN {X -29.5786,Y -38.6671,Z 64,A -132.0968,B 24.8738,C -2.5925,E1 24.9062,E2 -504.3458} C_DIS
LIN {X -26.4449,Y -40.8743,Z 64,A -128.1925,B 24.8754,C -2.5761,E1 24.9152,E2 -508.2238} C_DIS
LIN {X -23.8556,Y -42.4375,Z 64,A -123.8917,B 24.8748,C -2.5828,E1 24.9257,E2 -512.5534} C_DIS
LIN {X -20.0043,Y -44.3829,Z 64,A -119.5657,B 24.8765,C -2.565,E1 24.9365,E2 -516.8481} C_DIS
LIN {X -17.8319,Y -45.2993,Z 64,A -116.6496,B 24.8765,C -2.5645,E1 24.944,E2 -519.7695} C_DIS
LIN {X -14.8959,Y -46.348,Z 64,A -113.3758,B 24.8774,C -2.5552,E1 24.9526,E2 -523.0274} C_DIS
Enddeposition()
END
